LIN {X 0,Y 573.113,Z 1074.431,A -85,B 0,C 180,E1 -2244.193,E2 -2244.193} C_VEL
LIN {X 0,Y 573.004,Z 1079.986,A -85,B 0,C 180,E1 -2245.075,E2 -2245.075} C_VEL
LIN {X 0,Y 573.024,Z 1085.147,A -85,B 0,C 180,E1 -2246.132,E2 -2246.132} C_VEL
LIN {X 0,Y 572.99,Z 1087.788,A -85,B 0,C 180,E1 -2246.836,E2 -2246.836} C_VEL
LIN {X 0,Y 572.94,Z 1090.68,A -85,B 0,C 180,E1 -2247.891,E2 -2247.891} C_VEL
LIN {X 0,Y 572.944,Z 1091.936,A -85,B 0,C 180,E1 -2248.594,E2 -2248.594} C_VEL
LIN {X 0,Y 572.937,Z 1092.712,A -85,B 0,C 180,E1 -2249.297,E2 -2249.297} C_VEL
LIN {X 0,Y 572.935,Z 1093,A -85,B 0,C 180,E1 -2250,E2 -2250} C_VEL
LIN {X 0,Y 572.937,Z 1092.712,A -85,B 0,C 180,E1 -2250.703,E2 -2250.703} C_VEL
LIN {X 0,Y 572.944,Z 1091.936,A -85,B 0,C 180,E1 -2251.406,E2 -2251.406} C_VEL
LIN {X 0,Y 572.94,Z 1090.68,A -85,B 0,C 180,E1 -2252.109,E2 -2252.109} C_VEL
LIN {X 0,Y 572.99,Z 1087.788,A -85,B 0,C 180,E1 -2253.164,E2 -2253.164} C_VEL
LIN {X 0,Y 573.036,Z 1085.148,A -85,B 0,C 180,E1 -2253.868,E2 -2253.868} C_VEL
LIN {X 0,Y 573.004,Z 1079.986,A -85,B 0,C 180,E1 -2254.925,E2 -2254.925} C_VEL
LIN {X 0,Y 573.112,Z 1074.431,A -85,B 0,C 180,E1 -2255.806,E2 -2255.806} C_VEL
LIN {X 0,Y 573.155,Z 1067.55,A -85,B 0,C 180,E1 -2256.677,E2 -2256.677} C_VEL
LIN {X 0,Y 573.187,Z 1059.42,A -85,B 0,C 180,E1 -2257.485,E2 -2257.485} C_VEL
LIN {X 0,Y 573.256,Z 1051.769,A -85,B 0,C 180,E1 -2258.105,E2 -2258.105} C_VEL
LIN {X 0,Y 573.361,Z 1043.729,A -85,B 0,C 180,E1 -2258.636,E2 -2258.636} C_VEL
LIN {X 0,Y 573.393,Z 1035.4,A -85,B 0,C 180,E1 -2259.08,E2 -2259.08} C_VEL
LIN {X 0,Y 573.442,Z 1026.896,A -85,B 0,C 180,E1 -2259.434,E2 -2259.434} C_VEL
LIN {X 0,Y 573.468,Z 1016.757,A -85,B 0,C 180,E1 -2259.746,E2 -2259.746} C_VEL
LIN {X 0,Y 573.603,Z 1005.066,A -85,B 0,C 180,E1 -2259.966,E2 -2259.966} C_VEL
LIN {X 0,Y 573.476,Z 935.024,A -85,B 0,C 180,E1 -2260.842,E2 -2260.842} C_VEL
LIN {X 0,Y 573.182,Z 932.72,A -85,B 0,C 180,E1 -2260.883,E2 -2260.883} C_VEL
LIN {X 0,Y 573.294,Z 914.402,A -85,B 0,C 180,E1 -2263.83,E2 -2263.83} C_VEL
LIN {X 0,Y 573.477,Z 896.612,A -85,B 0,C 180,E1 -2266.725,E2 -2266.725} C_VEL
LIN {X 0,Y 573.619,Z 878.673,A -85,B 0,C 180,E1 -2269.69,E2 -2269.69} C_VEL
LIN {X 0,Y 573.625,Z 866.389,A -85,B 0,C 180,E1 -2271.754,E2 -2271.754} C_VEL
LIN {X 0,Y 573.2,Z 863.899,A -85,B 0,C 180,E1 -2272.197,E2 -2272.197} C_VEL
LIN {X 0,Y 573.186,Z 863.903,A -85,B 0,C 180,E1 -2274.861,E2 -2274.861} C_VEL
LIN {X 0,Y 573.182,Z 863.903,A -85,B 0,C 180,E1 -2276.979,E2 -2276.979} C_VEL
LIN {X 0,Y 573.193,Z 863.898,A -85,B 0,C 180,E1 -2279.479,E2 -2279.479} C_VEL
LIN {X 0,Y 573.218,Z 863.889,A -85,B 0,C 180,E1 -2282.223,E2 -2282.223} C_VEL
LIN {X 0,Y 573.212,Z 863.891,A -85,B 0,C 180,E1 -2284.768,E2 -2284.768} C_VEL
LIN {X 0,Y 573.184,Z 863.9,A -85,B 0,C 180,E1 -2287.812,E2 -2287.812} C_VEL
LIN {X 0,Y 573.197,Z 863.891,A -85,B 0,C 180,E1 -2290.529,E2 -2290.529} C_VEL
LIN {X 0,Y 573.183,Z 863.896,A -85,B 0,C 180,E1 -2293.364,E2 -2293.364} C_VEL
LIN {X 0,Y 573.191,Z 863.896,A -85,B 0,C 180,E1 -2296.337,E2 -2296.337} C_VEL
LIN {X 0,Y 573.183,Z 863.896,A -85,B 0,C 180,E1 -2298.539,E2 -2298.539} C_VEL
LIN {X 0,Y 573.174,Z 863.894,A -85,B 0,C 180,E1 -2301.293,E2 -2301.293} C_VEL
LIN {X 0,Y 573.178,Z 863.899,A -85,B 0,C 180,E1 -2304.023,E2 -2304.023} C_VEL
LIN {X 0,Y 573.22,Z 863.898,A -85,B 0,C 180,E1 -2306.515,E2 -2306.515} C_VEL
LIN {X 0,Y 573.198,Z 863.893,A -85,B 0,C 180,E1 -2309.123,E2 -2309.123} C_VEL
LIN {X 0,Y 573.19,Z 863.893,A -85,B 0,C 180,E1 -2311.983,E2 -2311.983} C_VEL
LIN {X 0,Y 573.194,Z 863.899,A -85,B 0,C 180,E1 -2314.587,E2 -2314.587} C_VEL
LIN {X 0,Y 573.191,Z 863.904,A -85,B 0,C 180,E1 -2316.899,E2 -2316.899} C_VEL
LIN {X 0,Y 573.223,Z 863.897,A -85,B 0,C 180,E1 -2319.173,E2 -2319.173} C_VEL
LIN {X 0,Y 573.189,Z 863.9,A -85,B 0,C 180,E1 -2321.41,E2 -2321.41} C_VEL
LIN {X 0,Y 573.247,Z 863.914,A -85,B 0,C 180,E1 -2322.52,E2 -2322.52} C_VEL
LIN {X 0,Y 573.186,Z 877.285,A -85,B 0,C 180,E1 -2325.444,E2 -2325.444} C_VEL
LIN {X 0,Y 573.114,Z 890.643,A -85,B 0,C 180,E1 -2328.327,E2 -2328.327} C_VEL
LIN {X 0,Y 573.113,Z 894.661,A -85,B 0,C 180,E1 -2329.188,E2 -2329.188} C_VEL
LIN {X 0,Y 573.677,Z 900.915,A -85,B 0,C 180,E1 -2329.281,E2 -2329.281} C_VEL
LIN {X 0,Y 573.529,Z 970.436,A -85,B 0,C 180,E1 -2330.167,E2 -2330.167} C_VEL
LIN {X 0,Y 573.478,Z 980.906,A -85,B 0,C 180,E1 -2330.411,E2 -2330.411} C_VEL
LIN {X 0,Y 573.381,Z 992.584,A -85,B 0,C 180,E1 -2330.832,E2 -2330.832} C_VEL
LIN {X 0,Y 573.369,Z 1003.02,A -85,B 0,C 180,E1 -2331.365,E2 -2331.365} C_VEL
LIN {X 0,Y 573.243,Z 1012.409,A -85,B 0,C 180,E1 -2331.984,E2 -2331.984} C_VEL
LIN {X 0,Y 573.188,Z 1021.892,A -85,B 0,C 180,E1 -2332.78,E2 -2332.78} C_VEL
LIN {X 0,Y 573.129,Z 1030.032,A -85,B 0,C 180,E1 -2333.664,E2 -2333.664} C_VEL
LIN {X 0,Y 573.051,Z 1036.508,A -85,B 0,C 180,E1 -2334.546,E2 -2334.546} C_VEL
LIN {X 0,Y 573.047,Z 1041.68,A -85,B 0,C 180,E1 -2335.428,E2 -2335.428} C_VEL
LIN {X 0,Y 573.025,Z 1046.439,A -85,B 0,C 180,E1 -2336.485,E2 -2336.485} C_VEL
LIN {X 0,Y 572.962,Z 1048.797,A -85,B 0,C 180,E1 -2337.188,E2 -2337.188} C_VEL
LIN {X 0,Y 572.94,Z 1050.597,A -85,B 0,C 180,E1 -2337.891,E2 -2337.891} C_VEL
LIN {X 0,Y 572.944,Z 1051.898,A -85,B 0,C 180,E1 -2338.595,E2 -2338.595} C_VEL
LIN {X 0,Y 572.936,Z 1052.709,A -85,B 0,C 180,E1 -2339.297,E2 -2339.297} C_VEL
LIN {X 0,Y 572.936,Z 1052.996,A -85,B 0,C 180,E1 -2340,E2 -2340} C_VEL
LIN {X 0,Y 572.937,Z 1052.75,A -85,B 0,C 180,E1 -2340.703,E2 -2340.703} C_VEL
LIN {X 0,Y 572.945,Z 1052.018,A -85,B 0,C 180,E1 -2341.406,E2 -2341.406} C_VEL
LIN {X 0,Y 572.941,Z 1050.801,A -85,B 0,C 180,E1 -2342.109,E2 -2342.109} C_VEL
LIN {X 0,Y 572.991,Z 1047.951,A -85,B 0,C 180,E1 -2343.164,E2 -2343.164} C_VEL
LIN {X 0,Y 573.033,Z 1043.853,A -85,B 0,C 180,E1 -2344.22,E2 -2344.22} C_VEL
LIN {X 0,Y 573.016,Z 1038.249,A -85,B 0,C 180,E1 -2345.278,E2 -2345.278} C_VEL
LIN {X 0,Y 573.145,Z 1032.173,A -85,B 0,C 180,E1 -2346.16,E2 -2346.16} C_VEL
LIN {X 0,Y 573.164,Z 1024.503,A -85,B 0,C 180,E1 -2347.044,E2 -2347.044} C_VEL
LIN {X 0,Y 573.237,Z 1015.883,A -85,B 0,C 180,E1 -2347.84,E2 -2347.84} C_VEL
LIN {X 0,Y 573.354,Z 1006.003,A -85,B 0,C 180,E1 -2348.548,E2 -2348.548} C_VEL
LIN {X 0,Y 573.379,Z 996.339,A -85,B 0,C 180,E1 -2349.08,E2 -2349.08} C_VEL
LIN {X 0,Y 573.411,Z 988.108,A -85,B 0,C 180,E1 -2349.435,E2 -2349.435} C_VEL
LIN {X 0,Y 573.475,Z 979.257,A -85,B 0,C 180,E1 -2349.724,E2 -2349.724} C_VEL
LIN {X 0,Y 573.546,Z 970.451,A -85,B 0,C 180,E1 -2349.923,E2 -2349.923} C_VEL
LIN {X 0,Y 573.521,Z 897.598,A -85,B 0,C 180,E1 -2350.854,E2 -2350.854} C_VEL
LIN {X 0,Y 573.113,Z 894.647,A -85,B 0,C 180,E1 -2350.905,E2 -2350.905} C_VEL
LIN {X 0,Y 573.165,Z 881.032,A -85,B 0,C 180,E1 -2353.834,E2 -2353.834} C_VEL
LIN {X 0,Y 573.155,Z 880.165,A -85,B 0,C 180,E1 -2354.022,E2 -2354.022} C_VEL
LIN {X 0,Y 572.495,Z 877.772,A -85,B 0,C 180,E1 -2354.558,E2 -2354.558} C_VEL
LIN {X 0,Y 566.909,Z 870.416,A -85,B 0,C 180,E1 -2356.327,E2 -2356.327} C_VEL
LIN {X 0,Y 566.259,Z 868.043,A -85,B 0,C 180,E1 -2356.873,E2 -2356.873} C_VEL
LIN {X 0,Y 566.195,Z 864.767,A -85,B 0,C 180,E1 -2357.612,E2 -2357.612} C_VEL
LIN {X 0,Y 566.151,Z 864.769,A -85,B 0,C 180,E1 -2360.34,E2 -2360.34} C_VEL
LIN {X 0,Y 566.132,Z 864.773,A -85,B 0,C 180,E1 -2362.634,E2 -2362.634} C_VEL
LIN {X 0,Y 566.164,Z 864.773,A -85,B 0,C 180,E1 -2365.018,E2 -2365.018} C_VEL
LIN {X 0,Y 566.161,Z 864.778,A -85,B 0,C 180,E1 -2367.342,E2 -2367.342} C_VEL
LIN {X 0,Y 566.147,Z 864.775,A -85,B 0,C 180,E1 -2369.772,E2 -2369.772} C_VEL
LIN {X 0,Y 566.176,Z 864.766,A -85,B 0,C 180,E1 -2372.425,E2 -2372.425} C_VEL
LIN {X 0,Y 566.162,Z 864.768,A -85,B 0,C 180,E1 -2374.987,E2 -2374.987} C_VEL
LIN {X 0,Y 566.181,Z 864.77,A -85,B 0,C 180,E1 -2377.463,E2 -2377.463} C_VEL
LIN {X 0,Y 566.159,Z 864.774,A -85,B 0,C 180,E1 -2380.204,E2 -2380.204} C_VEL
LIN {X 0,Y 566.144,Z 864.769,A -85,B 0,C 180,E1 -2383.06,E2 -2383.06} C_VEL
LIN {X 0,Y 566.146,Z 864.778,A -85,B 0,C 180,E1 -2386.055,E2 -2386.055} C_VEL
LIN {X 0,Y 566.135,Z 864.773,A -85,B 0,C 180,E1 -2388.857,E2 -2388.857} C_VEL
LIN {X 0,Y 566.158,Z 864.768,A -85,B 0,C 180,E1 -2391.449,E2 -2391.449} C_VEL
LIN {X 0,Y 566.159,Z 864.768,A -85,B 0,C 180,E1 -2393.793,E2 -2393.793} C_VEL
LIN {X 0,Y 566.198,Z 864.767,A -85,B 0,C 180,E1 -2396.269,E2 -2396.269} C_VEL
LIN {X 0,Y 566.172,Z 864.774,A -85,B 0,C 180,E1 -2398.928,E2 -2398.928} C_VEL
LIN {X 0,Y 566.143,Z 864.77,A -85,B 0,C 180,E1 -2401.854,E2 -2401.854} C_VEL
LIN {X 0,Y 566.171,Z 864.767,A -85,B 0,C 180,E1 -2404.249,E2 -2404.249} C_VEL
LIN {X 0,Y 566.149,Z 864.776,A -85,B 0,C 180,E1 -2407.367,E2 -2407.367} C_VEL
LIN {X 0,Y 566.159,Z 864.772,A -85,B 0,C 180,E1 -2409.661,E2 -2409.661} C_VEL
LIN {X 0,Y 566.164,Z 864.769,A -85,B 0,C 180,E1 -2411.921,E2 -2411.921} C_VEL
LIN {X 0,Y 566.182,Z 864.767,A -85,B 0,C 180,E1 -2414.89,E2 -2414.89} C_VEL
LIN {X 0,Y 566.159,Z 864.775,A -85,B 0,C 180,E1 -2417.817,E2 -2417.817} C_VEL
LIN {X 0,Y 566.132,Z 864.777,A -85,B 0,C 180,E1 -2419.991,E2 -2419.991} C_VEL
LIN {X 0,Y 566.183,Z 864.769,A -85,B 0,C 180,E1 -2422.152,E2 -2422.152} C_VEL
LIN {X 0,Y 566.247,Z 864.757,A -85,B 0,C 180,E1 -2425.016,E2 -2425.016} C_VEL
LIN {X 0,Y 566.279,Z 864.76,A -85,B 0,C 180,E1 -2427.866,E2 -2427.866} C_VEL
LIN {X 0,Y 566.288,Z 864.76,A -85,B 0,C 180,E1 -2430,E2 -2430} C_VEL
LIN {X 0,Y 566.239,Z 864.76,A -85,B 0,C 180,E1 -2432.846,E2 -2432.846} C_VEL
LIN {X 0,Y 566.222,Z 864.761,A -85,B 0,C 180,E1 -2435.699,E2 -2435.699} C_VEL
LIN {X 0,Y 566.187,Z 864.774,A -85,B 0,C 180,E1 -2438.567,E2 -2438.567} C_VEL
LIN {X 0,Y 566.194,Z 864.764,A -85,B 0,C 180,E1 -2441.455,E2 -2441.455} C_VEL
LIN {X 0,Y 566.18,Z 864.771,A -85,B 0,C 180,E1 -2444.482,E2 -2444.482} C_VEL
LIN {X 0,Y 566.174,Z 864.77,A -85,B 0,C 180,E1 -2447.333,E2 -2447.333} C_VEL
LIN {X 0,Y 566.175,Z 864.768,A -85,B 0,C 180,E1 -2449.582,E2 -2449.582} C_VEL
LIN {X 0,Y 566.143,Z 864.77,A -85,B 0,C 180,E1 -2451.865,E2 -2451.865} C_VEL
LIN {X 0,Y 566.149,Z 864.769,A -85,B 0,C 180,E1 -2454.183,E2 -2454.183} C_VEL
LIN {X 0,Y 566.17,Z 864.767,A -85,B 0,C 180,E1 -2456.65,E2 -2456.65} C_VEL
LIN {X 0,Y 566.149,Z 864.774,A -85,B 0,C 180,E1 -2459.772,E2 -2459.772} C_VEL
LIN {X 0,Y 566.141,Z 864.77,A -85,B 0,C 180,E1 -2462.419,E2 -2462.419} C_VEL
LIN {X 0,Y 566.163,Z 864.768,A -85,B 0,C 180,E1 -2464.986,E2 -2464.986} C_VEL
LIN {X 0,Y 566.158,Z 864.773,A -85,B 0,C 180,E1 -2467.464,E2 -2467.464} C_VEL
LIN {X 0,Y 566.161,Z 864.773,A -85,B 0,C 180,E1 -2470.203,E2 -2470.203} C_VEL
LIN {X 0,Y 566.143,Z 864.769,A -85,B 0,C 180,E1 -2473.06,E2 -2473.06} C_VEL
LIN {X 0,Y 566.146,Z 864.778,A -85,B 0,C 180,E1 -2476.055,E2 -2476.055} C_VEL
LIN {X 0,Y 566.136,Z 864.773,A -85,B 0,C 180,E1 -2478.856,E2 -2478.856} C_VEL
LIN {X 0,Y 566.158,Z 864.768,A -85,B 0,C 180,E1 -2481.449,E2 -2481.449} C_VEL
LIN {X 0,Y 566.138,Z 864.777,A -85,B 0,C 180,E1 -2484.306,E2 -2484.306} C_VEL
LIN {X 0,Y 566.165,Z 864.774,A -85,B 0,C 180,E1 -2486.894,E2 -2486.894} C_VEL
LIN {X 0,Y 566.151,Z 864.77,A -85,B 0,C 180,E1 -2489.405,E2 -2489.405} C_VEL
LIN {X 0,Y 566.143,Z 864.77,A -85,B 0,C 180,E1 -2491.853,E2 -2491.853} C_VEL
LIN {X 0,Y 566.171,Z 864.767,A -85,B 0,C 180,E1 -2494.248,E2 -2494.248} C_VEL
LIN {X 0,Y 566.148,Z 864.776,A -85,B 0,C 180,E1 -2497.367,E2 -2497.367} C_VEL
LIN {X 0,Y 566.157,Z 864.771,A -85,B 0,C 180,E1 -2499.66,E2 -2499.66} C_VEL
LIN {X 0,Y 566.163,Z 864.769,A -85,B 0,C 180,E1 -2501.92,E2 -2501.92} C_VEL
LIN {X 0,Y 566.174,Z 864.766,A -85,B 0,C 180,E1 -2504.151,E2 -2504.151} C_VEL
LIN {X 0,Y 566.157,Z 864.768,A -85,B 0,C 180,E1 -2506.357,E2 -2506.357} C_VEL
LIN {X 0,Y 566.199,Z 864.767,A -85,B 0,C 180,E1 -2509.269,E2 -2509.269} C_VEL
LIN {X 0,Y 566.181,Z 864.769,A -85,B 0,C 180,E1 -2512.152,E2 -2512.152} C_VEL
LIN {X 0,Y 566.246,Z 864.757,A -85,B 0,C 180,E1 -2515.015,E2 -2515.015} C_VEL
LIN {X 0,Y 566.278,Z 864.761,A -85,B 0,C 180,E1 -2517.866,E2 -2517.866} C_VEL
LIN {X 0,Y 566.286,Z 864.761,A -85,B 0,C 180,E1 -2520,E2 -2520} C_VEL
LIN {X 0,Y 566.237,Z 864.76,A -85,B 0,C 180,E1 -2522.845,E2 -2522.845} C_VEL
LIN {X 0,Y 566.22,Z 864.761,A -85,B 0,C 180,E1 -2525.698,E2 -2525.698} C_VEL
LIN {X 0,Y 566.184,Z 864.774,A -85,B 0,C 180,E1 -2528.566,E2 -2528.566} C_VEL
LIN {X 0,Y 566.191,Z 864.764,A -85,B 0,C 180,E1 -2531.455,E2 -2531.455} C_VEL
LIN {X 0,Y 566.205,Z 864.768,A -85,B 0,C 180,E1 -2534.493,E2 -2534.493} C_VEL
LIN {X 0,Y 566.171,Z 864.77,A -85,B 0,C 180,E1 -2537.332,E2 -2537.332} C_VEL
LIN {X 0,Y 566.171,Z 864.768,A -85,B 0,C 180,E1 -2539.582,E2 -2539.582} C_VEL
LIN {X 0,Y 566.14,Z 864.77,A -85,B 0,C 180,E1 -2541.864,E2 -2541.864} C_VEL
LIN {X 0,Y 566.146,Z 864.769,A -85,B 0,C 180,E1 -2544.183,E2 -2544.183} C_VEL
LIN {X 0,Y 566.166,Z 864.768,A -85,B 0,C 180,E1 -2546.65,E2 -2546.65} C_VEL
LIN {X 0,Y 566.145,Z 864.774,A -85,B 0,C 180,E1 -2549.772,E2 -2549.772} C_VEL
LIN {X 0,Y 566.137,Z 864.77,A -85,B 0,C 180,E1 -2552.419,E2 -2552.419} C_VEL
LIN {X 0,Y 566.16,Z 864.768,A -85,B 0,C 180,E1 -2554.986,E2 -2554.986} C_VEL
LIN {X 0,Y 566.156,Z 864.773,A -85,B 0,C 180,E1 -2557.464,E2 -2557.464} C_VEL
LIN {X 0,Y 566.157,Z 864.773,A -85,B 0,C 180,E1 -2560.203,E2 -2560.203} C_VEL
LIN {X 0,Y 566.141,Z 864.77,A -85,B 0,C 180,E1 -2563.06,E2 -2563.06} C_VEL
LIN {X 0,Y 566.143,Z 864.779,A -85,B 0,C 180,E1 -2566.054,E2 -2566.054} C_VEL
LIN {X 0,Y 566.132,Z 864.773,A -85,B 0,C 180,E1 -2568.856,E2 -2568.856} C_VEL
LIN {X 0,Y 566.155,Z 864.768,A -85,B 0,C 180,E1 -2571.449,E2 -2571.449} C_VEL
LIN {X 0,Y 566.135,Z 864.778,A -85,B 0,C 180,E1 -2574.306,E2 -2574.306} C_VEL
LIN {X 0,Y 566.16,Z 864.774,A -85,B 0,C 180,E1 -2576.894,E2 -2576.894} C_VEL
LIN {X 0,Y 566.147,Z 864.77,A -85,B 0,C 180,E1 -2579.405,E2 -2579.405} C_VEL
LIN {X 0,Y 566.138,Z 864.77,A -85,B 0,C 180,E1 -2581.853,E2 -2581.853} C_VEL
LIN {X 0,Y 566.167,Z 864.769,A -85,B 0,C 180,E1 -2584.248,E2 -2584.248} C_VEL
LIN {X 0,Y 566.155,Z 864.778,A -85,B 0,C 180,E1 -2587.367,E2 -2587.367} C_VEL
LIN {X 0,Y 566.203,Z 864.991,A -85,B 0,C 180,E1 -2587.706,E2 -2587.706} C_VEL
LIN {X 0,Y 566.808,Z 870.505,A -85,B 0,C 180,E1 -2588.675,E2 -2588.675} C_VEL
LIN {X 0,Y 566.569,Z 887.602,A -85,B 0,C 180,E1 -2591.56,E2 -2591.56} C_VEL
LIN {X 0,Y 566.37,Z 905.467,A -85,B 0,C 180,E1 -2594.526,E2 -2594.526} C_VEL
LIN {X 0,Y 566.196,Z 924.449,A -85,B 0,C 180,E1 -2597.636,E2 -2597.636} C_VEL
LIN {X 0,Y 566.143,Z 932.732,A -85,B 0,C 180,E1 -2598.982,E2 -2598.982} C_VEL
LIN {X 0,Y 566.664,Z 939.256,A -85,B 0,C 180,E1 -2599.08,E2 -2599.08} C_VEL
LIN {X 0,Y 566.574,Z 1009.129,A -85,B 0,C 180,E1 -2599.977,E2 -2599.977} C_VEL
LIN {X 0,Y 566.483,Z 1018.407,A -85,B 0,C 180,E1 -2600.178,E2 -2600.178} C_VEL
LIN {X 0,Y 566.455,Z 1026.888,A -85,B 0,C 180,E1 -2600.448,E2 -2600.448} C_VEL
LIN {X 0,Y 566.38,Z 1035.396,A -85,B 0,C 180,E1 -2600.807,E2 -2600.807} C_VEL
LIN {X 0,Y 566.346,Z 1043.727,A -85,B 0,C 180,E1 -2601.256,E2 -2601.256} C_VEL
LIN {X 0,Y 566.232,Z 1051.764,A -85,B 0,C 180,E1 -2601.794,E2 -2601.794} C_VEL
LIN {X 0,Y 566.146,Z 1059.414,A -85,B 0,C 180,E1 -2602.421,E2 -2602.421} C_VEL
LIN {X 0,Y 566.095,Z 1068.155,A -85,B 0,C 180,E1 -2603.309,E2 -2603.309} C_VEL
LIN {X 0,Y 566.057,Z 1074.432,A -85,B 0,C 180,E1 -2604.121,E2 -2604.121} C_VEL
LIN {X 0,Y 565.911,Z 1079.986,A -85,B 0,C 180,E1 -2605.013,E2 -2605.013} C_VEL
LIN {X 0,Y 565.934,Z 1085.147,A -85,B 0,C 180,E1 -2606.083,E2 -2606.083} C_VEL
LIN {X 0,Y 565.914,Z 1087.788,A -85,B 0,C 180,E1 -2606.796,E2 -2606.796} C_VEL
LIN {X 0,Y 565.841,Z 1090.68,A -85,B 0,C 180,E1 -2607.864,E2 -2607.864} C_VEL
LIN {X 0,Y 565.844,Z 1091.936,A -85,B 0,C 180,E1 -2608.576,E2 -2608.576} C_VEL
LIN {X 0,Y 565.837,Z 1092.711,A -85,B 0,C 180,E1 -2609.288,E2 -2609.288} C_VEL
LIN {X 0,Y 565.836,Z 1093,A -85,B 0,C 180,E1 -2610,E2 -2610} C_VEL
LIN {X 0,Y 565.837,Z 1092.711,A -85,B 0,C 180,E1 -2610.712,E2 -2610.712} C_VEL
LIN {X 0,Y 565.844,Z 1091.936,A -85,B 0,C 180,E1 -2611.423,E2 -2611.423} C_VEL
LIN {X 0,Y 565.84,Z 1090.681,A -85,B 0,C 180,E1 -2612.135,E2 -2612.135} C_VEL
LIN {X 0,Y 565.912,Z 1087.788,A -85,B 0,C 180,E1 -2613.204,E2 -2613.204} C_VEL
LIN {X 0,Y 565.944,Z 1085.148,A -85,B 0,C 180,E1 -2613.916,E2 -2613.916} C_VEL
LIN {X 0,Y 565.911,Z 1079.986,A -85,B 0,C 180,E1 -2614.987,E2 -2614.987} C_VEL
LIN {X 0,Y 566.082,Z 1073.188,A -85,B 0,C 180,E1 -2616.058,E2 -2616.058} C_VEL
LIN {X 0,Y 566.091,Z 1066.178,A -85,B 0,C 180,E1 -2616.907,E2 -2616.907} C_VEL
LIN {X 0,Y 566.145,Z 1058.407,A -85,B 0,C 180,E1 -2617.669,E2 -2617.669} C_VEL
LIN {X 0,Y 566.239,Z 1050.549,A -85,B 0,C 180,E1 -2618.296,E2 -2618.296} C_VEL
LIN {X 0,Y 566.354,Z 1040.735,A -85,B 0,C 180,E1 -2618.923,E2 -2618.923} C_VEL
LIN {X 0,Y 566.413,Z 1029.303,A -85,B 0,C 180,E1 -2619.463,E2 -2619.463} C_VEL
LIN {X 0,Y 566.505,Z 1019.249,A -85,B 0,C 180,E1 -2619.799,E2 -2619.799} C_VEL
LIN {X 0,Y 566.551,Z 1010.449,A -85,B 0,C 180,E1 -2620.001,E2 -2620.001} C_VEL
LIN {X 0,Y 566.645,Z 954.982,A -85,B 0,C 180,E1 -2620.722,E2 -2620.722} C_VEL
LIN {X 0,Y 566.639,Z 936.596,A -85,B 0,C 180,E1 -2620.954,E2 -2620.954} C_VEL
LIN {X 0,Y 566.146,Z 932.717,A -85,B 0,C 180,E1 -2621.02,E2 -2621.02} C_VEL
LIN {X 0,Y 566.268,Z 915.518,A -85,B 0,C 180,E1 -2623.822,E2 -2623.822} C_VEL
LIN {X 0,Y 566.439,Z 898.77,A -85,B 0,C 180,E1 -2626.581,E2 -2626.581} C_VEL
LIN {X 0,Y 566.664,Z 881.914,A -85,B 0,C 180,E1 -2629.394,E2 -2629.394} C_VEL
LIN {X 0,Y 566.77,Z 869.11,A -85,B 0,C 180,E1 -2631.564,E2 -2631.564} C_VEL
LIN {X 0,Y 566.178,Z 864.775,A -85,B 0,C 180,E1 -2632.343,E2 -2632.343} C_VEL
LIN {X 0,Y 566.139,Z 864.782,A -85,B 0,C 180,E1 -2635.013,E2 -2635.013} C_VEL
LIN {X 0,Y 566.155,Z 864.776,A -85,B 0,C 180,E1 -2637.342,E2 -2637.342} C_VEL
LIN {X 0,Y 566.142,Z 864.773,A -85,B 0,C 180,E1 -2639.772,E2 -2639.772} C_VEL
LIN {X 0,Y 566.169,Z 864.767,A -85,B 0,C 180,E1 -2642.424,E2 -2642.424} C_VEL
LIN {X 0,Y 566.158,Z 864.772,A -85,B 0,C 180,E1 -2644.986,E2 -2644.986} C_VEL
LIN {X 0,Y 566.152,Z 864.778,A -85,B 0,C 180,E1 -2647.464,E2 -2647.464} C_VEL
LIN {X 0,Y 566.154,Z 864.771,A -85,B 0,C 180,E1 -2650.204,E2 -2650.204} C_VEL
LIN {X 0,Y 566.135,Z 864.772,A -85,B 0,C 180,E1 -2653.06,E2 -2653.06} C_VEL
LIN {X 0,Y 566.142,Z 864.779,A -85,B 0,C 180,E1 -2656.055,E2 -2656.055} C_VEL
LIN {X 0,Y 566.131,Z 864.772,A -85,B 0,C 180,E1 -2658.857,E2 -2658.857} C_VEL
LIN {X 0,Y 566.158,Z 864.769,A -85,B 0,C 180,E1 -2661.449,E2 -2661.449} C_VEL
LIN {X 0,Y 566.133,Z 864.782,A -85,B 0,C 180,E1 -2664.306,E2 -2664.306} C_VEL
LIN {X 0,Y 566.159,Z 864.772,A -85,B 0,C 180,E1 -2666.894,E2 -2666.894} C_VEL
LIN {X 0,Y 566.145,Z 864.77,A -85,B 0,C 180,E1 -2669.405,E2 -2669.405} C_VEL
LIN {X 0,Y 566.137,Z 864.771,A -85,B 0,C 180,E1 -2671.854,E2 -2671.854} C_VEL
LIN {X 0,Y 566.166,Z 864.77,A -85,B 0,C 180,E1 -2674.249,E2 -2674.249} C_VEL
LIN {X 0,Y 566.144,Z 864.779,A -85,B 0,C 180,E1 -2676.725,E2 -2676.725} C_VEL
LIN {X 0,Y 566.187,Z 864.775,A -85,B 0,C 180,E1 -2678.902,E2 -2678.902} C_VEL
LIN {X 0,Y 566.165,Z 864.778,A -85,B 0,C 180,E1 -2681.171,E2 -2681.171} C_VEL
LIN {X 0,Y 566.232,Z 864.961,A -85,B 0,C 180,E1 -2682.53,E2 -2682.53} C_VEL
LIN {X 0,Y 566.156,Z 877.448,A -85,B 0,C 180,E1 -2685.294,E2 -2685.294} C_VEL
LIN {X 0,Y 566.053,Z 890.646,A -85,B 0,C 180,E1 -2688.179,E2 -2688.179} C_VEL
LIN {X 0,Y 566.052,Z 894.641,A -85,B 0,C 180,E1 -2689.047,E2 -2689.047} C_VEL
LIN {X 0,Y 566.699,Z 901.636,A -85,B 0,C 180,E1 -2689.156,E2 -2689.156} C_VEL
LIN {X 0,Y 566.557,Z 969.17,A -85,B 0,C 180,E1 -2690.022,E2 -2690.022} C_VEL
LIN {X 0,Y 566.515,Z 978.439,A -85,B 0,C 180,E1 -2690.224,E2 -2690.224} C_VEL
LIN {X 0,Y 566.408,Z 988.116,A -85,B 0,C 180,E1 -2690.538,E2 -2690.538} C_VEL
LIN {X 0,Y 566.411,Z 998.199,A -85,B 0,C 180,E1 -2690.988,E2 -2690.988} C_VEL
LIN {X 0,Y 566.282,Z 1008.722,A -85,B 0,C 180,E1 -2691.615,E2 -2691.615} C_VEL
LIN {X 0,Y 566.167,Z 1017.924,A -85,B 0,C 180,E1 -2692.332,E2 -2692.332} C_VEL
LIN {X 0,Y 566.101,Z 1025.875,A -85,B 0,C 180,E1 -2693.103,E2 -2693.103} C_VEL
LIN {X 0,Y 566.057,Z 1034.151,A -85,B 0,C 180,E1 -2694.121,E2 -2694.121} C_VEL
LIN {X 0,Y 565.912,Z 1039.765,A -85,B 0,C 180,E1 -2695.013,E2 -2695.013} C_VEL
LIN {X 0,Y 565.944,Z 1044.992,A -85,B 0,C 180,E1 -2696.084,E2 -2696.084} C_VEL
LIN {X 0,Y 565.881,Z 1048.799,A -85,B 0,C 180,E1 -2697.153,E2 -2697.153} C_VEL
LIN {X 0,Y 565.841,Z 1050.603,A -85,B 0,C 180,E1 -2697.865,E2 -2697.865} C_VEL
LIN {X 0,Y 565.843,Z 1051.904,A -85,B 0,C 180,E1 -2698.577,E2 -2698.577} C_VEL
LIN {X 0,Y 565.837,Z 1052.712,A -85,B 0,C 180,E1 -2699.289,E2 -2699.289} C_VEL
LIN {X 0,Y 565.837,Z 1052.996,A -85,B 0,C 180,E1 -2700,E2 -2700} C_VEL
LIN {X 0,Y 565.838,Z 1052.754,A -85,B 0,C 180,E1 -2700.712,E2 -2700.712} C_VEL
LIN {X 0,Y 565.845,Z 1052.022,A -85,B 0,C 180,E1 -2701.424,E2 -2701.424} C_VEL
LIN {X 0,Y 565.841,Z 1050.804,A -85,B 0,C 180,E1 -2702.136,E2 -2702.136} C_VEL
LIN {X 0,Y 565.913,Z 1047.953,A -85,B 0,C 180,E1 -2703.204,E2 -2703.204} C_VEL
LIN {X 0,Y 565.963,Z 1043.854,A -85,B 0,C 180,E1 -2704.273,E2 -2704.273} C_VEL
LIN {X 0,Y 565.946,Z 1038.246,A -85,B 0,C 180,E1 -2705.344,E2 -2705.344} C_VEL
LIN {X 0,Y 566.084,Z 1032.171,A -85,B 0,C 180,E1 -2706.237,E2 -2706.237} C_VEL
LIN {X 0,Y 566.116,Z 1024.503,A -85,B 0,C 180,E1 -2707.132,E2 -2707.132} C_VEL
LIN {X 0,Y 566.175,Z 1015.878,A -85,B 0,C 180,E1 -2707.938,E2 -2707.938} C_VEL
LIN {X 0,Y 566.328,Z 1006.002,A -85,B 0,C 180,E1 -2708.654,E2 -2708.654} C_VEL
LIN {X 0,Y 566.365,Z 996.332,A -85,B 0,C 180,E1 -2709.194,E2 -2709.194} C_VEL
LIN {X 0,Y 566.447,Z 986.892,A -85,B 0,C 180,E1 -2709.598,E2 -2709.598} C_VEL
LIN {X 0,Y 566.506,Z 976.737,A -85,B 0,C 180,E1 -2709.912,E2 -2709.912} C_VEL
LIN {X 0,Y 566.596,Z 965.018,A -85,B 0,C 180,E1 -2710.136,E2 -2710.136} C_VEL
LIN {X 0,Y 566.639,Z 898.908,A -85,B 0,C 180,E1 -2710.97,E2 -2710.97} C_VEL
LIN {X 0,Y 566.045,Z 894.625,A -85,B 0,C 180,E1 -2711.047,E2 -2711.047} C_VEL
LIN {X 0,Y 566.118,Z 880.858,A -85,B 0,C 180,E1 -2714.047,E2 -2714.047} C_VEL
LIN {X 0,Y 566.259,Z 868.043,A -85,B 0,C 180,E1 -2716.873,E2 -2716.873} C_VEL
LIN {X 0,Y 565.931,Z 866.698,A -85,B 0,C 180,E1 -2717.242,E2 -2717.242} C_VEL
LIN {X 0,Y 564.573,Z 865.564,A -85,B 0,C 180,E1 -2717.812,E2 -2717.812} C_VEL
LIN {X 0,Y 562.707,Z 865.21,A -85,B 0,C 180,E1 -2718.385,E2 -2718.385} C_VEL
LIN {X 0,Y 560.273,Z 865.509,A -85,B 0,C 180,E1 -2719.175,E2 -2719.175} C_VEL
LIN {X 0,Y 559.217,Z 865.638,A -85,B 0,C 180,E1 -2719.783,E2 -2719.783} C_VEL
LIN {X 0,Y 559.123,Z 865.644,A -85,B 0,C 180,E1 -2719.989,E2 -2719.989} C_VEL
LIN {X 0,Y 559.098,Z 865.647,A -85,B 0,C 180,E1 -2722.155,E2 -2722.155} C_VEL
LIN {X 0,Y 559.131,Z 865.652,A -85,B 0,C 180,E1 -2725.176,E2 -2725.176} C_VEL
LIN {X 0,Y 559.101,Z 865.652,A -85,B 0,C 180,E1 -2727.717,E2 -2727.717} C_VEL
LIN {X 0,Y 559.093,Z 865.649,A -85,B 0,C 180,E1 -2730.187,E2 -2730.187} C_VEL
LIN {X 0,Y 559.135,Z 865.643,A -85,B 0,C 180,E1 -2732.717,E2 -2732.717} C_VEL
LIN {X 0,Y 559.115,Z 865.649,A -85,B 0,C 180,E1 -2735.326,E2 -2735.326} C_VEL
LIN {X 0,Y 559.115,Z 865.653,A -85,B 0,C 180,E1 -2738.02,E2 -2738.02} C_VEL
LIN {X 0,Y 559.093,Z 865.648,A -85,B 0,C 180,E1 -2740.819,E2 -2740.819} C_VEL
LIN {X 0,Y 559.1,Z 865.652,A -85,B 0,C 180,E1 -2743.739,E2 -2743.739} C_VEL
LIN {X 0,Y 559.093,Z 865.658,A -85,B 0,C 180,E1 -2746.261,E2 -2746.261} C_VEL
LIN {X 0,Y 559.092,Z 865.648,A -85,B 0,C 180,E1 -2749.182,E2 -2749.182} C_VEL
LIN {X 0,Y 559.099,Z 865.65,A -85,B 0,C 180,E1 -2751.98,E2 -2751.98} C_VEL
LIN {X 0,Y 559.121,Z 865.652,A -85,B 0,C 180,E1 -2754.79,E2 -2754.79} C_VEL
LIN {X 0,Y 559.138,Z 865.643,A -85,B 0,C 180,E1 -2757.368,E2 -2757.368} C_VEL
LIN {X 0,Y 559.098,Z 865.648,A -85,B 0,C 180,E1 -2760.153,E2 -2760.153} C_VEL
LIN {X 0,Y 559.114,Z 865.652,A -85,B 0,C 180,E1 -2763.185,E2 -2763.185} C_VEL
LIN {X 0,Y 559.089,Z 865.652,A -85,B 0,C 180,E1 -2765.492,E2 -2765.492} C_VEL
LIN {X 0,Y 559.14,Z 865.643,A -85,B 0,C 180,E1 -2768.456,E2 -2768.456} C_VEL
LIN {X 0,Y 559.138,Z 865.647,A -85,B 0,C 180,E1 -2770.925,E2 -2770.925} C_VEL
LIN {X 0,Y 559.136,Z 865.645,A -85,B 0,C 180,E1 -2773.947,E2 -2773.947} C_VEL
LIN {X 0,Y 559.145,Z 865.643,A -85,B 0,C 180,E1 -2776.184,E2 -2776.184} C_VEL
LIN {X 0,Y 559.158,Z 865.642,A -85,B 0,C 180,E1 -2779.133,E2 -2779.133} C_VEL
LIN {X 0,Y 559.138,Z 865.649,A -85,B 0,C 180,E1 -2782.053,E2 -2782.053} C_VEL
LIN {X 0,Y 559.224,Z 865.632,A -85,B 0,C 180,E1 -2784.953,E2 -2784.953} C_VEL
LIN {X 0,Y 559.249,Z 865.635,A -85,B 0,C 180,E1 -2787.84,E2 -2787.84} C_VEL
LIN {X 0,Y 559.256,Z 865.636,A -85,B 0,C 180,E1 -2790,E2 -2790} C_VEL
LIN {X 0,Y 559.206,Z 865.635,A -85,B 0,C 180,E1 -2792.882,E2 -2792.882} C_VEL
LIN {X 0,Y 559.193,Z 865.637,A -85,B 0,C 180,E1 -2795.771,E2 -2795.771} C_VEL
LIN {X 0,Y 559.152,Z 865.649,A -85,B 0,C 180,E1 -2798.675,E2 -2798.675} C_VEL
LIN {X 0,Y 559.134,Z 865.643,A -85,B 0,C 180,E1 -2801.602,E2 -2801.602} C_VEL
LIN {X 0,Y 559.138,Z 865.649,A -85,B 0,C 180,E1 -2804.568,E2 -2804.568} C_VEL
LIN {X 0,Y 559.123,Z 865.646,A -85,B 0,C 180,E1 -2807.558,E2 -2807.558} C_VEL
LIN {X 0,Y 559.138,Z 865.643,A -85,B 0,C 180,E1 -2809.839,E2 -2809.839} C_VEL
LIN {X 0,Y 559.1,Z 865.647,A -85,B 0,C 180,E1 -2812.155,E2 -2812.155} C_VEL
LIN {X 0,Y 559.122,Z 865.654,A -85,B 0,C 180,E1 -2815.173,E2 -2815.173} C_VEL
LIN {X 0,Y 559.103,Z 865.652,A -85,B 0,C 180,E1 -2817.717,E2 -2817.717} C_VEL
LIN {X 0,Y 559.095,Z 865.648,A -85,B 0,C 180,E1 -2820.187,E2 -2820.187} C_VEL
LIN {X 0,Y 559.1,Z 865.647,A -85,B 0,C 180,E1 -2822.719,E2 -2822.719} C_VEL
LIN {X 0,Y 559.117,Z 865.649,A -85,B 0,C 180,E1 -2825.325,E2 -2825.325} C_VEL
LIN {X 0,Y 559.094,Z 865.655,A -85,B 0,C 180,E1 -2828.021,E2 -2828.021} C_VEL
LIN {X 0,Y 559.094,Z 865.648,A -85,B 0,C 180,E1 -2830.818,E2 -2830.818} C_VEL
LIN {X 0,Y 559.095,Z 865.653,A -85,B 0,C 180,E1 -2833.739,E2 -2833.739} C_VEL
LIN {X 0,Y 559.093,Z 865.657,A -85,B 0,C 180,E1 -2836.261,E2 -2836.261} C_VEL
LIN {X 0,Y 559.093,Z 865.648,A -85,B 0,C 180,E1 -2839.181,E2 -2839.181} C_VEL
LIN {X 0,Y 559.093,Z 865.651,A -85,B 0,C 180,E1 -2841.979,E2 -2841.979} C_VEL
LIN {X 0,Y 559.121,Z 865.651,A -85,B 0,C 180,E1 -2844.789,E2 -2844.789} C_VEL
LIN {X 0,Y 559.139,Z 865.643,A -85,B 0,C 180,E1 -2847.368,E2 -2847.368} C_VEL
LIN {X 0,Y 559.098,Z 865.649,A -85,B 0,C 180,E1 -2850.152,E2 -2850.152} C_VEL
LIN {X 0,Y 559.114,Z 865.652,A -85,B 0,C 180,E1 -2853.185,E2 -2853.185} C_VEL
LIN {X 0,Y 559.089,Z 865.652,A -85,B 0,C 180,E1 -2855.491,E2 -2855.491} C_VEL
LIN {X 0,Y 559.14,Z 865.643,A -85,B 0,C 180,E1 -2858.456,E2 -2858.456} C_VEL
LIN {X 0,Y 559.137,Z 865.647,A -85,B 0,C 180,E1 -2860.925,E2 -2860.925} C_VEL
LIN {X 0,Y 559.144,Z 865.649,A -85,B 0,C 180,E1 -2863.196,E2 -2863.196} C_VEL
LIN {X 0,Y 559.14,Z 865.643,A -85,B 0,C 180,E1 -2866.183,E2 -2866.183} C_VEL
LIN {X 0,Y 559.157,Z 865.643,A -85,B 0,C 180,E1 -2869.132,E2 -2869.132} C_VEL
LIN {X 0,Y 559.136,Z 865.648,A -85,B 0,C 180,E1 -2872.052,E2 -2872.052} C_VEL
LIN {X 0,Y 559.222,Z 865.632,A -85,B 0,C 180,E1 -2874.953,E2 -2874.953} C_VEL
LIN {X 0,Y 559.248,Z 865.636,A -85,B 0,C 180,E1 -2877.839,E2 -2877.839} C_VEL
LIN {X 0,Y 559.254,Z 865.636,A -85,B 0,C 180,E1 -2880,E2 -2880} C_VEL
LIN {X 0,Y 559.204,Z 865.636,A -85,B 0,C 180,E1 -2882.881,E2 -2882.881} C_VEL
LIN {X 0,Y 559.191,Z 865.637,A -85,B 0,C 180,E1 -2885.77,E2 -2885.77} C_VEL
LIN {X 0,Y 559.15,Z 865.649,A -85,B 0,C 180,E1 -2888.675,E2 -2888.675} C_VEL
LIN {X 0,Y 559.131,Z 865.643,A -85,B 0,C 180,E1 -2891.602,E2 -2891.602} C_VEL
LIN {X 0,Y 559.155,Z 865.647,A -85,B 0,C 180,E1 -2894.576,E2 -2894.576} C_VEL
LIN {X 0,Y 559.12,Z 865.646,A -85,B 0,C 180,E1 -2897.558,E2 -2897.558} C_VEL
LIN {X 0,Y 559.135,Z 865.643,A -85,B 0,C 180,E1 -2899.838,E2 -2899.838} C_VEL
LIN {X 0,Y 559.097,Z 865.647,A -85,B 0,C 180,E1 -2902.154,E2 -2902.154} C_VEL
LIN {X 0,Y 559.118,Z 865.655,A -85,B 0,C 180,E1 -2905.173,E2 -2905.173} C_VEL
LIN {X 0,Y 559.099,Z 865.652,A -85,B 0,C 180,E1 -2907.716,E2 -2907.716} C_VEL
LIN {X 0,Y 559.091,Z 865.649,A -85,B 0,C 180,E1 -2910.186,E2 -2910.186} C_VEL
LIN {X 0,Y 559.096,Z 865.648,A -85,B 0,C 180,E1 -2912.719,E2 -2912.719} C_VEL
LIN {X 0,Y 559.113,Z 865.65,A -85,B 0,C 180,E1 -2915.325,E2 -2915.325} C_VEL
LIN {X 0,Y 559.094,Z 865.655,A -85,B 0,C 180,E1 -2918.02,E2 -2918.02} C_VEL
LIN {X 0,Y 559.09,Z 865.648,A -85,B 0,C 180,E1 -2920.818,E2 -2920.818} C_VEL
LIN {X 0,Y 559.097,Z 865.653,A -85,B 0,C 180,E1 -2923.738,E2 -2923.738} C_VEL
LIN {X 0,Y 559.09,Z 865.657,A -85,B 0,C 180,E1 -2926.261,E2 -2926.261} C_VEL
LIN {X 0,Y 559.089,Z 865.648,A -85,B 0,C 180,E1 -2929.181,E2 -2929.181} C_VEL
LIN {X 0,Y 559.089,Z 865.652,A -85,B 0,C 180,E1 -2931.979,E2 -2931.979} C_VEL
LIN {X 0,Y 559.117,Z 865.651,A -85,B 0,C 180,E1 -2934.789,E2 -2934.789} C_VEL
LIN {X 0,Y 559.134,Z 865.644,A -85,B 0,C 180,E1 -2937.368,E2 -2937.368} C_VEL
LIN {X 0,Y 559.094,Z 865.649,A -85,B 0,C 180,E1 -2940.152,E2 -2940.152} C_VEL
LIN {X 0,Y 559.11,Z 865.654,A -85,B 0,C 180,E1 -2943.185,E2 -2943.185} C_VEL
LIN {X 0,Y 559.086,Z 865.655,A -85,B 0,C 180,E1 -2945.491,E2 -2945.491} C_VEL
LIN {X 0,Y 559.153,Z 865.829,A -85,B 0,C 180,E1 -2947.556,E2 -2947.556} C_VEL
LIN {X 0,Y 559.866,Z 870.486,A -85,B 0,C 180,E1 -2948.395,E2 -2948.395} C_VEL
LIN {X 0,Y 559.597,Z 887.602,A -85,B 0,C 180,E1 -2951.321,E2 -2951.321} C_VEL
LIN {X 0,Y 559.365,Z 904.351,A -85,B 0,C 180,E1 -2954.141,E2 -2954.141} C_VEL
LIN {X 0,Y 559.163,Z 922.216,A -85,B 0,C 180,E1 -2957.109,E2 -2957.109} C_VEL
LIN {X 0,Y 559.115,Z 932.672,A -85,B 0,C 180,E1 -2958.832,E2 -2958.832} C_VEL
LIN {X 0,Y 559.707,Z 939.696,A -85,B 0,C 180,E1 -2958.948,E2 -2958.948} C_VEL
LIN {X 0,Y 559.598,Z 1009.129,A -85,B 0,C 180,E1 -2959.85,E2 -2959.85} C_VEL
LIN {X 0,Y 559.497,Z 1018.407,A -85,B 0,C 180,E1 -2960.054,E2 -2960.054} C_VEL
LIN {X 0,Y 559.472,Z 1026.887,A -85,B 0,C 180,E1 -2960.327,E2 -2960.327} C_VEL
LIN {X 0,Y 559.379,Z 1035.397,A -85,B 0,C 180,E1 -2960.691,E2 -2960.691} C_VEL
LIN {X 0,Y 559.328,Z 1043.728,A -85,B 0,C 180,E1 -2961.146,E2 -2961.146} C_VEL
LIN {X 0,Y 559.184,Z 1051.766,A -85,B 0,C 180,E1 -2961.689,E2 -2961.689} C_VEL
LIN {X 0,Y 559.094,Z 1060.428,A -85,B 0,C 180,E1 -2962.415,E2 -2962.415} C_VEL
LIN {X 0,Y 559.031,Z 1068.753,A -85,B 0,C 180,E1 -2963.299,E2 -2963.299} C_VEL
LIN {X 0,Y 559.004,Z 1074.432,A -85,B 0,C 180,E1 -2964.046,E2 -2964.046} C_VEL
LIN {X 0,Y 558.825,Z 1079.987,A -85,B 0,C 180,E1 -2964.949,E2 -2964.949} C_VEL
LIN {X 0,Y 558.851,Z 1085.147,A -85,B 0,C 180,E1 -2966.034,E2 -2966.034} C_VEL
LIN {X 0,Y 558.84,Z 1087.788,A -85,B 0,C 180,E1 -2966.756,E2 -2966.756} C_VEL
LIN {X 0,Y 558.746,Z 1090.681,A -85,B 0,C 180,E1 -2967.837,E2 -2967.837} C_VEL
LIN {X 0,Y 558.744,Z 1091.935,A -85,B 0,C 180,E1 -2968.558,E2 -2968.558} C_VEL
LIN {X 0,Y 558.737,Z 1092.71,A -85,B 0,C 180,E1 -2969.279,E2 -2969.279} C_VEL
LIN {X 0,Y 558.737,Z 1093,A -85,B 0,C 180,E1 -2970,E2 -2970} C_VEL
LIN {X 0,Y 558.737,Z 1092.71,A -85,B 0,C 180,E1 -2970.721,E2 -2970.721} C_VEL
LIN {X 0,Y 558.744,Z 1091.935,A -85,B 0,C 180,E1 -2971.441,E2 -2971.441} C_VEL
LIN {X 0,Y 558.746,Z 1090.681,A -85,B 0,C 180,E1 -2972.162,E2 -2972.162} C_VEL
LIN {X 0,Y 558.835,Z 1087.788,A -85,B 0,C 180,E1 -2973.244,E2 -2973.244} C_VEL
LIN {X 0,Y 558.859,Z 1085.148,A -85,B 0,C 180,E1 -2973.966,E2 -2973.966} C_VEL
LIN {X 0,Y 558.825,Z 1079.986,A -85,B 0,C 180,E1 -2975.05,E2 -2975.05} C_VEL
LIN {X 0,Y 559.018,Z 1073.188,A -85,B 0,C 180,E1 -2976.134,E2 -2976.134} C_VEL
LIN {X 0,Y 559.035,Z 1065.746,A -85,B 0,C 180,E1 -2977.04,E2 -2977.04} C_VEL
LIN {X 0,Y 559.118,Z 1058.408,A -85,B 0,C 180,E1 -2977.766,E2 -2977.766} C_VEL
LIN {X 0,Y 559.223,Z 1050.548,A -85,B 0,C 180,E1 -2978.401,E2 -2978.401} C_VEL
LIN {X 0,Y 559.318,Z 1040.733,A -85,B 0,C 180,E1 -2979.037,E2 -2979.037} C_VEL
LIN {X 0,Y 559.43,Z 1029.304,A -85,B 0,C 180,E1 -2979.582,E2 -2979.582} C_VEL
LIN {X 0,Y 559.52,Z 1019.249,A -85,B 0,C 180,E1 -2979.923,E2 -2979.923} C_VEL
LIN {X 0,Y 559.561,Z 1010.448,A -85,B 0,C 180,E1 -2980.127,E2 -2980.127} C_VEL
LIN {X 0,Y 559.707,Z 963.925,A -85,B 0,C 180,E1 -2980.742,E2 -2980.742} C_VEL
LIN {X 0,Y 559.613,Z 936.673,A -85,B 0,C 180,E1 -2981.093,E2 -2981.093} C_VEL
LIN {X 0,Y 559.107,Z 932.701,A -85,B 0,C 180,E1 -2981.164,E2 -2981.164} C_VEL
LIN {X 0,Y 559.244,Z 915.518,A -85,B 0,C 180,E1 -2983.999,E2 -2983.999} C_VEL
LIN {X 0,Y 559.474,Z 897.223,A -85,B 0,C 180,E1 -2987.054,E2 -2987.054} C_VEL
LIN {X 0,Y 559.73,Z 879.788,A -85,B 0,C 180,E1 -2990.008,E2 -2990.008} C_VEL
LIN {X 0,Y 559.701,Z 869.021,A -85,B 0,C 180,E1 -2991.866,E2 -2991.866} C_VEL
LIN {X 0,Y 559.131,Z 865.653,A -85,B 0,C 180,E1 -2992.494,E2 -2992.494} C_VEL
LIN {X 0,Y 559.097,Z 865.656,A -85,B 0,C 180,E1 -2995.302,E2 -2995.302} C_VEL
LIN {X 0,Y 559.097,Z 865.651,A -85,B 0,C 180,E1 -2997.717,E2 -2997.717} C_VEL
LIN {X 0,Y 559.089,Z 865.649,A -85,B 0,C 180,E1 -3000.187,E2 -3000.187} C_VEL
LIN {X 0,Y 559.13,Z 865.646,A -85,B 0,C 180,E1 -3002.717,E2 -3002.717} C_VEL
LIN {X 0,Y 559.111,Z 865.655,A -85,B 0,C 180,E1 -3005.325,E2 -3005.325} C_VEL
LIN {X 0,Y 559.088,Z 865.653,A -85,B 0,C 180,E1 -3008.021,E2 -3008.021} C_VEL
LIN {X 0,Y 559.087,Z 865.649,A -85,B 0,C 180,E1 -3010.819,E2 -3010.819} C_VEL
LIN {X 0,Y 559.087,Z 865.658,A -85,B 0,C 180,E1 -3013.739,E2 -3013.739} C_VEL
LIN {X 0,Y 559.089,Z 865.654,A -85,B 0,C 180,E1 -3016.261,E2 -3016.261} C_VEL
LIN {X 0,Y 559.088,Z 865.649,A -85,B 0,C 180,E1 -3019.182,E2 -3019.182} C_VEL
LIN {X 0,Y 559.092,Z 865.655,A -85,B 0,C 180,E1 -3021.979,E2 -3021.979} C_VEL
LIN {X 0,Y 559.116,Z 865.649,A -85,B 0,C 180,E1 -3024.79,E2 -3024.79} C_VEL
LIN {X 0,Y 559.133,Z 865.644,A -85,B 0,C 180,E1 -3027.368,E2 -3027.368} C_VEL
LIN {X 0,Y 559.093,Z 865.652,A -85,B 0,C 180,E1 -3030.153,E2 -3030.153} C_VEL
LIN {X 0,Y 559.107,Z 865.65,A -85,B 0,C 180,E1 -3033.186,E2 -3033.186} C_VEL
LIN {X 0,Y 559.084,Z 865.652,A -85,B 0,C 180,E1 -3035.492,E2 -3035.492} C_VEL
LIN {X 0,Y 559.154,Z 865.647,A -85,B 0,C 180,E1 -3038.623,E2 -3038.623} C_VEL
LIN {X 0,Y 559.133,Z 865.653,A -85,B 0,C 180,E1 -3040.925,E2 -3040.925} C_VEL
LIN {X 0,Y 559.168,Z 865.833,A -85,B 0,C 180,E1 -3042.499,E2 -3042.499} C_VEL
LIN {X 0,Y 559.125,Z 877.284,A -85,B 0,C 180,E1 -3045.068,E2 -3045.068} C_VEL
LIN {X 0,Y 558.994,Z 888.978,A -85,B 0,C 180,E1 -3047.659,E2 -3047.659} C_VEL
LIN {X 0,Y 558.996,Z 894.846,A -85,B 0,C 180,E1 -3048.917,E2 -3048.917} C_VEL
LIN {X 0,Y 559.741,Z 901.021,A -85,B 0,C 180,E1 -3049.011,E2 -3049.011} C_VEL
LIN {X 0,Y 559.583,Z 969.203,A -85,B 0,C 180,E1 -3049.896,E2 -3049.896} C_VEL
LIN {X 0,Y 559.53,Z 978.461,A -85,B 0,C 180,E1 -3050.101,E2 -3050.101} C_VEL
LIN {X 0,Y 559.414,Z 988.134,A -85,B 0,C 180,E1 -3050.418,E2 -3050.418} C_VEL
LIN {X 0,Y 559.383,Z 998.214,A -85,B 0,C 180,E1 -3050.874,E2 -3050.874} C_VEL
LIN {X 0,Y 559.266,Z 1008.726,A -85,B 0,C 180,E1 -3051.509,E2 -3051.509} C_VEL
LIN {X 0,Y 559.121,Z 1017.934,A -85,B 0,C 180,E1 -3052.234,E2 -3052.234} C_VEL
LIN {X 0,Y 559.068,Z 1025.368,A -85,B 0,C 180,E1 -3052.96,E2 -3052.96} C_VEL
LIN {X 0,Y 559.007,Z 1032.839,A -85,B 0,C 180,E1 -3053.866,E2 -3053.866} C_VEL
LIN {X 0,Y 558.826,Z 1039.767,A -85,B 0,C 180,E1 -3054.95,E2 -3054.95} C_VEL
LIN {X 0,Y 558.859,Z 1045,A -85,B 0,C 180,E1 -3056.034,E2 -3056.034} C_VEL
LIN {X 0,Y 558.804,Z 1048.802,A -85,B 0,C 180,E1 -3057.117,E2 -3057.117} C_VEL
LIN {X 0,Y 558.747,Z 1050.608,A -85,B 0,C 180,E1 -3057.838,E2 -3057.838} C_VEL
LIN {X 0,Y 558.743,Z 1051.909,A -85,B 0,C 180,E1 -3058.559,E2 -3058.559} C_VEL
LIN {X 0,Y 558.737,Z 1052.714,A -85,B 0,C 180,E1 -3059.28,E2 -3059.28} C_VEL
LIN {X 0,Y 558.738,Z 1052.996,A -85,B 0,C 180,E1 -3060,E2 -3060} C_VEL
LIN {X 0,Y 558.738,Z 1052.757,A -85,B 0,C 180,E1 -3060.721,E2 -3060.721} C_VEL
LIN {X 0,Y 558.745,Z 1052.026,A -85,B 0,C 180,E1 -3061.442,E2 -3061.442} C_VEL
LIN {X 0,Y 558.747,Z 1050.807,A -85,B 0,C 180,E1 -3062.163,E2 -3062.163} C_VEL
LIN {X 0,Y 558.836,Z 1047.955,A -85,B 0,C 180,E1 -3063.245,E2 -3063.245} C_VEL
LIN {X 0,Y 558.894,Z 1043.854,A -85,B 0,C 180,E1 -3064.327,E2 -3064.327} C_VEL
LIN {X 0,Y 558.881,Z 1038.242,A -85,B 0,C 180,E1 -3065.412,E2 -3065.412} C_VEL
LIN {X 0,Y 559.006,Z 1032.167,A -85,B 0,C 180,E1 -3066.316,E2 -3066.316} C_VEL
LIN {X 0,Y 559.056,Z 1024.502,A -85,B 0,C 180,E1 -3067.222,E2 -3067.222} C_VEL
LIN {X 0,Y 559.142,Z 1015.872,A -85,B 0,C 180,E1 -3068.039,E2 -3068.039} C_VEL
LIN {X 0,Y 559.32,Z 1006,A -85,B 0,C 180,E1 -3068.764,E2 -3068.764} C_VEL
LIN {X 0,Y 559.37,Z 996.324,A -85,B 0,C 180,E1 -3069.31,E2 -3069.31} C_VEL
LIN {X 0,Y 559.455,Z 986.876,A -85,B 0,C 180,E1 -3069.719,E2 -3069.719} C_VEL
LIN {X 0,Y 559.518,Z 976.714,A -85,B 0,C 180,E1 -3070.037,E2 -3070.037} C_VEL
LIN {X 0,Y 559.626,Z 964.973,A -85,B 0,C 180,E1 -3070.264,E2 -3070.264} C_VEL
LIN {X 0,Y 559.552,Z 898.727,A -85,B 0,C 180,E1 -3071.113,E2 -3071.113} C_VEL
LIN {X 0,Y 558.976,Z 894.639,A -85,B 0,C 180,E1 -3071.185,E2 -3071.185} C_VEL
LIN {X 0,Y 559.06,Z 882.698,A -85,B 0,C 180,E1 -3073.819,E2 -3073.819} C_VEL
LIN {X 0,Y 559.216,Z 868.846,A -85,B 0,C 180,E1 -3076.91,E2 -3076.91} C_VEL
LIN {X 0,Y 559.16,Z 865.643,A -85,B 0,C 180,E1 -3077.652,E2 -3077.652} C_VEL
LIN {X 0,Y 559.123,Z 865.644,A -85,B 0,C 180,E1 -3079.989,E2 -3079.989} C_VEL
LIN {X 0,Y 558.426,Z 865.735,A -85,B 0,C 180,E1 -3080.59,E2 -3080.59} C_VEL
LIN {X 0,Y 555.535,Z 866.095,A -85,B 0,C 180,E1 -3081.565,E2 -3081.565} C_VEL
LIN {X 0,Y 553.121,Z 866.394,A -85,B 0,C 180,E1 -3082.35,E2 -3082.35} C_VEL
LIN {X 0,Y 552.109,Z 866.525,A -85,B 0,C 180,E1 -3082.956,E2 -3082.956} C_VEL
LIN {X 0,Y 552.039,Z 866.535,A -85,B 0,C 180,E1 -3083.161,E2 -3083.161} C_VEL
LIN {X 0,Y 552.069,Z 866.528,A -85,B 0,C 180,E1 -3085.648,E2 -3085.648} C_VEL
LIN {X 0,Y 552.072,Z 866.523,A -85,B 0,C 180,E1 -3088.552,E2 -3088.552} C_VEL
LIN {X 0,Y 552.094,Z 866.529,A -85,B 0,C 180,E1 -3091.472,E2 -3091.472} C_VEL
LIN {X 0,Y 552.095,Z 866.523,A -85,B 0,C 180,E1 -3094.164,E2 -3094.164} C_VEL
LIN {X 0,Y 552.049,Z 866.525,A -85,B 0,C 180,E1 -3096.752,E2 -3096.752} C_VEL
LIN {X 0,Y 552.078,Z 866.526,A -85,B 0,C 180,E1 -3099.532,E2 -3099.532} C_VEL
LIN {X 0,Y 552.081,Z 866.526,A -85,B 0,C 180,E1 -3102.431,E2 -3102.431} C_VEL
LIN {X 0,Y 552.068,Z 866.525,A -85,B 0,C 180,E1 -3105.56,E2 -3105.56} C_VEL
LIN {X 0,Y 552.052,Z 866.532,A -85,B 0,C 180,E1 -3108.548,E2 -3108.548} C_VEL
LIN {X 0,Y 552.071,Z 866.523,A -85,B 0,C 180,E1 -3111.407,E2 -3111.407} C_VEL
LIN {X 0,Y 552.064,Z 866.534,A -85,B 0,C 180,E1 -3114.563,E2 -3114.563} C_VEL
LIN {X 0,Y 552.098,Z 866.523,A -85,B 0,C 180,E1 -3117.157,E2 -3117.157} C_VEL
LIN {X 0,Y 552.069,Z 866.523,A -85,B 0,C 180,E1 -3119.959,E2 -3119.959} C_VEL
LIN {X 0,Y 552.079,Z 866.531,A -85,B 0,C 180,E1 -3123.014,E2 -3123.014} C_VEL
LIN {X 0,Y 552.068,Z 866.523,A -85,B 0,C 180,E1 -3125.96,E2 -3125.96} C_VEL
LIN {X 0,Y 552.097,Z 866.529,A -85,B 0,C 180,E1 -3129.119,E2 -3129.119} C_VEL
LIN {X 0,Y 552.071,Z 866.531,A -85,B 0,C 180,E1 -3131.443,E2 -3131.443} C_VEL
LIN {X 0,Y 552.084,Z 866.526,A -85,B 0,C 180,E1 -3133.736,E2 -3133.736} C_VEL
LIN {X 0,Y 552.109,Z 866.521,A -85,B 0,C 180,E1 -3136.004,E2 -3136.004} C_VEL
LIN {X 0,Y 552.122,Z 866.517,A -85,B 0,C 180,E1 -3138.993,E2 -3138.993} C_VEL
LIN {X 0,Y 552.108,Z 866.526,A -85,B 0,C 180,E1 -3141.951,E2 -3141.951} C_VEL
LIN {X 0,Y 552.201,Z 866.506,A -85,B 0,C 180,E1 -3144.889,E2 -3144.889} C_VEL
LIN {X 0,Y 552.22,Z 866.511,A -85,B 0,C 180,E1 -3147.812,E2 -3147.812} C_VEL
LIN {X 0,Y 552.225,Z 866.512,A -85,B 0,C 180,E1 -3150,E2 -3150} C_VEL
LIN {X 0,Y 552.173,Z 866.511,A -85,B 0,C 180,E1 -3152.918,E2 -3152.918} C_VEL
LIN {X 0,Y 552.166,Z 866.513,A -85,B 0,C 180,E1 -3155.844,E2 -3155.844} C_VEL
LIN {X 0,Y 552.125,Z 866.522,A -85,B 0,C 180,E1 -3158.786,E2 -3158.786} C_VEL
LIN {X 0,Y 552.083,Z 866.521,A -85,B 0,C 180,E1 -3161.752,E2 -3161.752} C_VEL
LIN {X 0,Y 552.086,Z 866.529,A -85,B 0,C 180,E1 -3164.652,E2 -3164.652} C_VEL
LIN {X 0,Y 552.098,Z 866.523,A -85,B 0,C 180,E1 -3167.305,E2 -3167.305} C_VEL
LIN {X 0,Y 552.095,Z 866.52,A -85,B 0,C 180,E1 -3170.103,E2 -3170.103} C_VEL
LIN {X 0,Y 552.041,Z 866.527,A -85,B 0,C 180,E1 -3172.453,E2 -3172.453} C_VEL
LIN {X 0,Y 552.066,Z 866.533,A -85,B 0,C 180,E1 -3175.329,E2 -3175.329} C_VEL
LIN {X 0,Y 552.051,Z 866.526,A -85,B 0,C 180,E1 -3178.102,E2 -3178.102} C_VEL
LIN {X 0,Y 552.07,Z 866.523,A -85,B 0,C 180,E1 -3180.612,E2 -3180.612} C_VEL
LIN {X 0,Y 552.054,Z 866.529,A -85,B 0,C 180,E1 -3183.19,E2 -3183.19} C_VEL
LIN {X 0,Y 552.068,Z 866.532,A -85,B 0,C 180,E1 -3185.845,E2 -3185.845} C_VEL
LIN {X 0,Y 552.073,Z 866.523,A -85,B 0,C 180,E1 -3189.054,E2 -3189.054} C_VEL
LIN {X 0,Y 552.083,Z 866.525,A -85,B 0,C 180,E1 -3192.409,E2 -3192.409} C_VEL
LIN {X 0,Y 552.067,Z 866.525,A -85,B 0,C 180,E1 -3195.559,E2 -3195.559} C_VEL
LIN {X 0,Y 552.053,Z 866.531,A -85,B 0,C 180,E1 -3198.547,E2 -3198.547} C_VEL
LIN {X 0,Y 552.07,Z 866.523,A -85,B 0,C 180,E1 -3201.406,E2 -3201.406} C_VEL
LIN {X 0,Y 552.064,Z 866.534,A -85,B 0,C 180,E1 -3204.563,E2 -3204.563} C_VEL
LIN {X 0,Y 552.099,Z 866.522,A -85,B 0,C 180,E1 -3207.157,E2 -3207.157} C_VEL
LIN {X 0,Y 552.069,Z 866.523,A -85,B 0,C 180,E1 -3209.959,E2 -3209.959} C_VEL
LIN {X 0,Y 552.079,Z 866.531,A -85,B 0,C 180,E1 -3213.013,E2 -3213.013} C_VEL
LIN {X 0,Y 552.068,Z 866.523,A -85,B 0,C 180,E1 -3215.96,E2 -3215.96} C_VEL
LIN {X 0,Y 552.096,Z 866.529,A -85,B 0,C 180,E1 -3219.118,E2 -3219.118} C_VEL
LIN {X 0,Y 552.07,Z 866.531,A -85,B 0,C 180,E1 -3221.442,E2 -3221.442} C_VEL
LIN {X 0,Y 552.083,Z 866.526,A -85,B 0,C 180,E1 -3223.736,E2 -3223.736} C_VEL
LIN {X 0,Y 552.103,Z 866.521,A -85,B 0,C 180,E1 -3226.003,E2 -3226.003} C_VEL
LIN {X 0,Y 552.121,Z 866.518,A -85,B 0,C 180,E1 -3228.992,E2 -3228.992} C_VEL
LIN {X 0,Y 552.106,Z 866.526,A -85,B 0,C 180,E1 -3231.95,E2 -3231.95} C_VEL
LIN {X 0,Y 552.199,Z 866.507,A -85,B 0,C 180,E1 -3234.888,E2 -3234.888} C_VEL
LIN {X 0,Y 552.219,Z 866.511,A -85,B 0,C 180,E1 -3237.812,E2 -3237.812} C_VEL
LIN {X 0,Y 552.223,Z 866.512,A -85,B 0,C 180,E1 -3240,E2 -3240} C_VEL
LIN {X 0,Y 552.171,Z 866.511,A -85,B 0,C 180,E1 -3242.918,E2 -3242.918} C_VEL
LIN {X 0,Y 552.164,Z 866.513,A -85,B 0,C 180,E1 -3245.844,E2 -3245.844} C_VEL
LIN {X 0,Y 552.122,Z 866.522,A -85,B 0,C 180,E1 -3248.786,E2 -3248.786} C_VEL
LIN {X 0,Y 552.08,Z 866.522,A -85,B 0,C 180,E1 -3251.752,E2 -3251.752} C_VEL
LIN {X 0,Y 552.12,Z 866.527,A -85,B 0,C 180,E1 -3254.749,E2 -3254.749} C_VEL
LIN {X 0,Y 552.079,Z 866.522,A -85,B 0,C 180,E1 -3257.789,E2 -3257.789} C_VEL
LIN {X 0,Y 552.091,Z 866.52,A -85,B 0,C 180,E1 -3260.102,E2 -3260.102} C_VEL
LIN {X 0,Y 552.038,Z 866.528,A -85,B 0,C 180,E1 -3262.453,E2 -3262.453} C_VEL
LIN {X 0,Y 552.063,Z 866.533,A -85,B 0,C 180,E1 -3265.329,E2 -3265.329} C_VEL
LIN {X 0,Y 552.047,Z 866.526,A -85,B 0,C 180,E1 -3268.102,E2 -3268.102} C_VEL
LIN {X 0,Y 552.066,Z 866.523,A -85,B 0,C 180,E1 -3270.611,E2 -3270.611} C_VEL
LIN {X 0,Y 552.05,Z 866.529,A -85,B 0,C 180,E1 -3273.19,E2 -3273.19} C_VEL
LIN {X 0,Y 552.064,Z 866.532,A -85,B 0,C 180,E1 -3275.845,E2 -3275.845} C_VEL
LIN {X 0,Y 552.071,Z 866.523,A -85,B 0,C 180,E1 -3279.054,E2 -3279.054} C_VEL
LIN {X 0,Y 552.079,Z 866.526,A -85,B 0,C 180,E1 -3282.409,E2 -3282.409} C_VEL
LIN {X 0,Y 552.065,Z 866.525,A -85,B 0,C 180,E1 -3285.559,E2 -3285.559} C_VEL
LIN {X 0,Y 552.049,Z 866.531,A -85,B 0,C 180,E1 -3288.547,E2 -3288.547} C_VEL
LIN {X 0,Y 552.066,Z 866.523,A -85,B 0,C 180,E1 -3291.406,E2 -3291.406} C_VEL
LIN {X 0,Y 552.06,Z 866.534,A -85,B 0,C 180,E1 -3294.563,E2 -3294.563} C_VEL
LIN {X 0,Y 552.094,Z 866.522,A -85,B 0,C 180,E1 -3297.157,E2 -3297.157} C_VEL
LIN {X 0,Y 552.065,Z 866.524,A -85,B 0,C 180,E1 -3299.959,E2 -3299.959} C_VEL
LIN {X 0,Y 552.075,Z 866.533,A -85,B 0,C 180,E1 -3303.013,E2 -3303.013} C_VEL
LIN {X 0,Y 552.065,Z 866.527,A -85,B 0,C 180,E1 -3305.96,E2 -3305.96} C_VEL
LIN {X 0,Y 552.095,Z 866.666,A -85,B 0,C 180,E1 -3307.401,E2 -3307.401} C_VEL
LIN {X 0,Y 552.899,Z 871.97,A -85,B 0,C 180,E1 -3308.369,E2 -3308.369} C_VEL
LIN {X 0,Y 552.619,Z 887.602,A -85,B 0,C 180,E1 -3311.077,E2 -3311.077} C_VEL
LIN {X 0,Y 552.406,Z 903.234,A -85,B 0,C 180,E1 -3313.746,E2 -3313.746} C_VEL
LIN {X 0,Y 552.154,Z 921.099,A -85,B 0,C 180,E1 -3316.755,E2 -3316.755} C_VEL
LIN {X 0,Y 552.083,Z 932.723,A -85,B 0,C 180,E1 -3318.696,E2 -3318.696} C_VEL
LIN {X 0,Y 552.753,Z 940.071,A -85,B 0,C 180,E1 -3318.812,E2 -3318.812} C_VEL
LIN {X 0,Y 552.633,Z 1009.129,A -85,B 0,C 180,E1 -3319.721,E2 -3319.721} C_VEL
LIN {X 0,Y 552.497,Z 1018.406,A -85,B 0,C 180,E1 -3319.927,E2 -3319.927} C_VEL
LIN {X 0,Y 552.476,Z 1026.886,A -85,B 0,C 180,E1 -3320.204,E2 -3320.204} C_VEL
LIN {X 0,Y 552.385,Z 1035.395,A -85,B 0,C 180,E1 -3320.572,E2 -3320.572} C_VEL
LIN {X 0,Y 552.311,Z 1043.728,A -85,B 0,C 180,E1 -3321.032,E2 -3321.032} C_VEL
LIN {X 0,Y 552.162,Z 1051.767,A -85,B 0,C 180,E1 -3321.583,E2 -3321.583} C_VEL
LIN {X 0,Y 552.048,Z 1060.429,A -85,B 0,C 180,E1 -3322.318,E2 -3322.318} C_VEL
LIN {X 0,Y 551.953,Z 1069.431,A -85,B 0,C 180,E1 -3323.3,E2 -3323.3} C_VEL
LIN {X 0,Y 551.917,Z 1075.61,A -85,B 0,C 180,E1 -3324.153,E2 -3324.153} C_VEL
LIN {X 0,Y 551.746,Z 1079.987,A -85,B 0,C 180,E1 -3324.884,E2 -3324.884} C_VEL
LIN {X 0,Y 551.773,Z 1085.148,A -85,B 0,C 180,E1 -3325.983,E2 -3325.983} C_VEL
LIN {X 0,Y 551.766,Z 1087.788,A -85,B 0,C 180,E1 -3326.714,E2 -3326.714} C_VEL
LIN {X 0,Y 551.657,Z 1090.681,A -85,B 0,C 180,E1 -3327.81,E2 -3327.81} C_VEL
LIN {X 0,Y 551.643,Z 1091.934,A -85,B 0,C 180,E1 -3328.54,E2 -3328.54} C_VEL
LIN {X 0,Y 551.638,Z 1092.71,A -85,B 0,C 180,E1 -3329.27,E2 -3329.27} C_VEL
LIN {X 0,Y 551.637,Z 1093,A -85,B 0,C 180,E1 -3330,E2 -3330} C_VEL
LIN {X 0,Y 551.638,Z 1092.71,A -85,B 0,C 180,E1 -3330.73,E2 -3330.73} C_VEL
LIN {X 0,Y 551.643,Z 1091.935,A -85,B 0,C 180,E1 -3331.46,E2 -3331.46} C_VEL
LIN {X 0,Y 551.657,Z 1090.681,A -85,B 0,C 180,E1 -3332.19,E2 -3332.19} C_VEL
LIN {X 0,Y 551.761,Z 1087.788,A -85,B 0,C 180,E1 -3333.286,E2 -3333.286} C_VEL
LIN {X 0,Y 551.78,Z 1085.148,A -85,B 0,C 180,E1 -3334.017,E2 -3334.017} C_VEL
LIN {X 0,Y 551.745,Z 1079.986,A -85,B 0,C 180,E1 -3335.115,E2 -3335.115} C_VEL
LIN {X 0,Y 551.956,Z 1073.401,A -85,B 0,C 180,E1 -3336.184,E2 -3336.184} C_VEL
LIN {X 0,Y 551.992,Z 1065.745,A -85,B 0,C 180,E1 -3337.131,E2 -3337.131} C_VEL
LIN {X 0,Y 552.075,Z 1058.407,A -85,B 0,C 180,E1 -3337.865,E2 -3337.865} C_VEL
LIN {X 0,Y 552.197,Z 1050.546,A -85,B 0,C 180,E1 -3338.508,E2 -3338.508} C_VEL
LIN {X 0,Y 552.304,Z 1040.732,A -85,B 0,C 180,E1 -3339.152,E2 -3339.152} C_VEL
LIN {X 0,Y 552.451,Z 1029.305,A -85,B 0,C 180,E1 -3339.704,E2 -3339.704} C_VEL
LIN {X 0,Y 552.511,Z 1019.25,A -85,B 0,C 180,E1 -3340.05,E2 -3340.05} C_VEL
LIN {X 0,Y 552.577,Z 1010.448,A -85,B 0,C 180,E1 -3340.257,E2 -3340.257} C_VEL
LIN {X 0,Y 552.742,Z 969.291,A -85,B 0,C 180,E1 -3340.809,E2 -3340.809} C_VEL
LIN {X 0,Y 552.612,Z 937.019,A -85,B 0,C 180,E1 -3341.23,E2 -3341.23} C_VEL
LIN {X 0,Y 552.063,Z 932.72,A -85,B 0,C 180,E1 -3341.305,E2 -3341.305} C_VEL
LIN {X 0,Y 552.208,Z 915.545,A -85,B 0,C 180,E1 -3344.177,E2 -3344.177} C_VEL
LIN {X 0,Y 552.476,Z 898.77,A -85,B 0,C 180,E1 -3347.012,E2 -3347.012} C_VEL
LIN {X 0,Y 552.773,Z 880.904,A -85,B 0,C 180,E1 -3350.077,E2 -3350.077} C_VEL
LIN {X 0,Y 552.778,Z 870.712,A -85,B 0,C 180,E1 -3351.857,E2 -3351.857} C_VEL
LIN {X 0,Y 552.08,Z 866.532,A -85,B 0,C 180,E1 -3352.649,E2 -3352.649} C_VEL
LIN {X 0,Y 552.046,Z 866.53,A -85,B 0,C 180,E1 -3355.648,E2 -3355.648} C_VEL
LIN {X 0,Y 552.068,Z 866.526,A -85,B 0,C 180,E1 -3358.551,E2 -3358.551} C_VEL
LIN {X 0,Y 552.09,Z 866.529,A -85,B 0,C 180,E1 -3361.472,E2 -3361.472} C_VEL
LIN {X 0,Y 552.091,Z 866.522,A -85,B 0,C 180,E1 -3364.164,E2 -3364.164} C_VEL
LIN {X 0,Y 552.041,Z 866.527,A -85,B 0,C 180,E1 -3366.752,E2 -3366.752} C_VEL
LIN {X 0,Y 552.067,Z 866.533,A -85,B 0,C 180,E1 -3369.533,E2 -3369.533} C_VEL
LIN {X 0,Y 552.076,Z 866.524,A -85,B 0,C 180,E1 -3372.431,E2 -3372.431} C_VEL
LIN {X 0,Y 552.062,Z 866.529,A -85,B 0,C 180,E1 -3375.559,E2 -3375.559} C_VEL
LIN {X 0,Y 552.048,Z 866.529,A -85,B 0,C 180,E1 -3378.548,E2 -3378.548} C_VEL
LIN {X 0,Y 552.067,Z 866.524,A -85,B 0,C 180,E1 -3381.407,E2 -3381.407} C_VEL
LIN {X 0,Y 552.058,Z 866.531,A -85,B 0,C 180,E1 -3384.563,E2 -3384.563} C_VEL
LIN {X 0,Y 552.093,Z 866.522,A -85,B 0,C 180,E1 -3387.157,E2 -3387.157} C_VEL
LIN {X 0,Y 552.064,Z 866.526,A -85,B 0,C 180,E1 -3389.959,E2 -3389.959} C_VEL
LIN {X 0,Y 552.073,Z 866.529,A -85,B 0,C 180,E1 -3393.014,E2 -3393.014} C_VEL
LIN {X 0,Y 552.058,Z 866.527,A -85,B 0,C 180,E1 -3395.96,E2 -3395.96} C_VEL
LIN {X 0,Y 552.07,Z 866.533,A -85,B 0,C 180,E1 -3399.118,E2 -3399.118} C_VEL
LIN {X 0,Y 552.069,Z 866.532,A -85,B 0,C 180,E1 -3401.443,E2 -3401.443} C_VEL
LIN {X 0,Y 552.132,Z 866.673,A -85,B 0,C 180,E1 -3402.46,E2 -3402.46} C_VEL
LIN {X 0,Y 552.041,Z 878.957,A -85,B 0,C 180,E1 -3405.249,E2 -3405.249} C_VEL
LIN {X 0,Y 551.929,Z 892.322,A -85,B 0,C 180,E1 -3408.245,E2 -3408.245} C_VEL
LIN {X 0,Y 551.908,Z 894.629,A -85,B 0,C 180,E1 -3408.758,E2 -3408.758} C_VEL
LIN {X 0,Y 552.785,Z 902.281,A -85,B 0,C 180,E1 -3408.886,E2 -3408.886} C_VEL
LIN {X 0,Y 552.597,Z 969.236,A -85,B 0,C 180,E1 -3409.767,E2 -3409.767} C_VEL
LIN {X 0,Y 552.548,Z 978.481,A -85,B 0,C 180,E1 -3409.974,E2 -3409.974} C_VEL
LIN {X 0,Y 552.432,Z 988.152,A -85,B 0,C 180,E1 -3410.296,E2 -3410.296} C_VEL
LIN {X 0,Y 552.352,Z 998.23,A -85,B 0,C 180,E1 -3410.756,E2 -3410.756} C_VEL
LIN {X 0,Y 552.23,Z 1008.729,A -85,B 0,C 180,E1 -3411.4,E2 -3411.4} C_VEL
LIN {X 0,Y 552.077,Z 1017.945,A -85,B 0,C 180,E1 -3412.135,E2 -3412.135} C_VEL
LIN {X 0,Y 552.004,Z 1025.378,A -85,B 0,C 180,E1 -3412.87,E2 -3412.87} C_VEL
LIN {X 0,Y 551.932,Z 1033.053,A -85,B 0,C 180,E1 -3413.816,E2 -3413.816} C_VEL
LIN {X 0,Y 551.746,Z 1039.77,A -85,B 0,C 180,E1 -3414.885,E2 -3414.885} C_VEL
LIN {X 0,Y 551.78,Z 1045.008,A -85,B 0,C 180,E1 -3415.983,E2 -3415.983} C_VEL
LIN {X 0,Y 551.73,Z 1048.804,A -85,B 0,C 180,E1 -3417.08,E2 -3417.08} C_VEL
LIN {X 0,Y 551.657,Z 1050.613,A -85,B 0,C 180,E1 -3417.81,E2 -3417.81} C_VEL
LIN {X 0,Y 551.643,Z 1051.915,A -85,B 0,C 180,E1 -3418.54,E2 -3418.54} C_VEL
LIN {X 0,Y 551.638,Z 1052.715,A -85,B 0,C 180,E1 -3419.27,E2 -3419.27} C_VEL
LIN {X 0,Y 551.638,Z 1052.996,A -85,B 0,C 180,E1 -3420,E2 -3420} C_VEL
LIN {X 0,Y 551.639,Z 1052.76,A -85,B 0,C 180,E1 -3420.73,E2 -3420.73} C_VEL
LIN {X 0,Y 551.645,Z 1052.03,A -85,B 0,C 180,E1 -3421.46,E2 -3421.46} C_VEL
LIN {X 0,Y 551.658,Z 1050.809,A -85,B 0,C 180,E1 -3422.191,E2 -3422.191} C_VEL
LIN {X 0,Y 551.761,Z 1047.957,A -85,B 0,C 180,E1 -3423.286,E2 -3423.286} C_VEL
LIN {X 0,Y 551.806,Z 1043.852,A -85,B 0,C 180,E1 -3424.383,E2 -3424.383} C_VEL
LIN {X 0,Y 551.82,Z 1038.239,A -85,B 0,C 180,E1 -3425.482,E2 -3425.482} C_VEL
LIN {X 0,Y 551.926,Z 1031.878,A -85,B 0,C 180,E1 -3426.436,E2 -3426.436} C_VEL
LIN {X 0,Y 551.996,Z 1024.502,A -85,B 0,C 180,E1 -3427.315,E2 -3427.315} C_VEL
LIN {X 0,Y 552.104,Z 1015.866,A -85,B 0,C 180,E1 -3428.142,E2 -3428.142} C_VEL
LIN {X 0,Y 552.302,Z 1005.996,A -85,B 0,C 180,E1 -3428.876,E2 -3428.876} C_VEL
LIN {X 0,Y 552.359,Z 996.316,A -85,B 0,C 180,E1 -3429.429,E2 -3429.429} C_VEL
LIN {X 0,Y 552.449,Z 988.07,A -85,B 0,C 180,E1 -3429.797,E2 -3429.797} C_VEL
LIN {X 0,Y 552.525,Z 978.364,A -85,B 0,C 180,E1 -3430.119,E2 -3430.119} C_VEL
LIN {X 0,Y 552.627,Z 969.053,A -85,B 0,C 180,E1 -3430.326,E2 -3430.326} C_VEL
LIN {X 0,Y 552.636,Z 899.555,A -85,B 0,C 180,E1 -3431.242,E2 -3431.242} C_VEL
LIN {X 0,Y 551.94,Z 894.569,A -85,B 0,C 180,E1 -3431.344,E2 -3431.344} C_VEL
LIN {X 0,Y 552.004,Z 881.304,A -85,B 0,C 180,E1 -3434.313,E2 -3434.313} C_VEL
LIN {X 0,Y 552.204,Z 867.919,A -85,B 0,C 180,E1 -3437.343,E2 -3437.343} C_VEL
LIN {X 0,Y 552.135,Z 866.519,A -85,B 0,C 180,E1 -3437.719,E2 -3437.719} C_VEL
LIN {X 0,Y 552.092,Z 866.52,A -85,B 0,C 180,E1 -3440.103,E2 -3440.103} C_VEL
LIN {X 0,Y 552.039,Z 866.528,A -85,B 0,C 180,E1 -3442.454,E2 -3442.454} C_VEL
LIN {X 0,Y 552.039,Z 866.535,A -85,B 0,C 180,E1 -3443.161,E2 -3443.161} C_VEL
LIN {X 0,Y 551.403,Z 866.62,A -85,B 0,C 180,E1 -3443.771,E2 -3443.771} C_VEL
LIN {X 0,Y 548.559,Z 866.972,A -85,B 0,C 180,E1 -3444.76,E2 -3444.76} C_VEL
LIN {X 0,Y 546.139,Z 867.268,A -85,B 0,C 180,E1 -3445.556,E2 -3445.556} C_VEL
LIN {X 0,Y 545.105,Z 867.391,A -85,B 0,C 180,E1 -3446.171,E2 -3446.171} C_VEL
LIN {X 0,Y 545.024,Z 867.401,A -85,B 0,C 180,E1 -3446.379,E2 -3446.379} C_VEL
LIN {X 0,Y 545.012,Z 867.411,A -85,B 0,C 180,E1 -3449.342,E2 -3449.342} C_VEL
LIN {X 0,Y 545.041,Z 867.403,A -85,B 0,C 180,E1 -3451.916,E2 -3451.916} C_VEL
LIN {X 0,Y 545.046,Z 867.398,A -85,B 0,C 180,E1 -3454.566,E2 -3454.566} C_VEL
LIN {X 0,Y 545.008,Z 867.405,A -85,B 0,C 180,E1 -3457.307,E2 -3457.307} C_VEL
LIN {X 0,Y 545.008,Z 867.409,A -85,B 0,C 180,E1 -3460.148,E2 -3460.148} C_VEL
LIN {X 0,Y 545.018,Z 867.401,A -85,B 0,C 180,E1 -3463.113,E2 -3463.113} C_VEL
LIN {X 0,Y 545.026,Z 867.41,A -85,B 0,C 180,E1 -3466.23,E2 -3466.23} C_VEL
LIN {X 0,Y 544.995,Z 867.406,A -85,B 0,C 180,E1 -3468.877,E2 -3468.877} C_VEL
LIN {X 0,Y 545.021,Z 867.403,A -85,B 0,C 180,E1 -3471.869,E2 -3471.869} C_VEL
LIN {X 0,Y 545.024,Z 867.411,A -85,B 0,C 180,E1 -3474.531,E2 -3474.531} C_VEL
LIN {X 0,Y 545.053,Z 867.4,A -85,B 0,C 180,E1 -3477.211,E2 -3477.211} C_VEL
LIN {X 0,Y 545.019,Z 867.401,A -85,B 0,C 180,E1 -3479.808,E2 -3479.808} C_VEL
LIN {X 0,Y 545,Z 867.406,A -85,B 0,C 180,E1 -3482.339,E2 -3482.339} C_VEL
LIN {X 0,Y 545.023,Z 867.408,A -85,B 0,C 180,E1 -3484.816,E2 -3484.816} C_VEL
LIN {X 0,Y 545.01,Z 867.411,A -85,B 0,C 180,E1 -3487.241,E2 -3487.241} C_VEL
LIN {X 0,Y 545.092,Z 867.392,A -85,B 0,C 180,E1 -3490.257,E2 -3490.257} C_VEL
LIN {X 0,Y 545.054,Z 867.398,A -85,B 0,C 180,E1 -3492.749,E2 -3492.749} C_VEL
LIN {X 0,Y 545.069,Z 867.4,A -85,B 0,C 180,E1 -3495.819,E2 -3495.819} C_VEL
LIN {X 0,Y 545.07,Z 867.395,A -85,B 0,C 180,E1 -3498.848,E2 -3498.848} C_VEL
LIN {X 0,Y 545.066,Z 867.405,A -85,B 0,C 180,E1 -3501.846,E2 -3501.846} C_VEL
LIN {X 0,Y 545.159,Z 867.384,A -85,B 0,C 180,E1 -3504.823,E2 -3504.823} C_VEL
LIN {X 0,Y 545.191,Z 867.386,A -85,B 0,C 180,E1 -3507.784,E2 -3507.784} C_VEL
LIN {X 0,Y 545.193,Z 867.388,A -85,B 0,C 180,E1 -3510,E2 -3510} C_VEL
LIN {X 0,Y 545.141,Z 867.387,A -85,B 0,C 180,E1 -3512.956,E2 -3512.956} C_VEL
LIN {X 0,Y 545.119,Z 867.392,A -85,B 0,C 180,E1 -3515.92,E2 -3515.92} C_VEL
LIN {X 0,Y 545.068,Z 867.4,A -85,B 0,C 180,E1 -3518.901,E2 -3518.901} C_VEL
LIN {X 0,Y 545.056,Z 867.397,A -85,B 0,C 180,E1 -3521.906,E2 -3521.906} C_VEL
LIN {X 0,Y 545.04,Z 867.407,A -85,B 0,C 180,E1 -3524.945,E2 -3524.945} C_VEL
LIN {X 0,Y 545.049,Z 867.398,A -85,B 0,C 180,E1 -3528.027,E2 -3528.027} C_VEL
LIN {X 0,Y 545.033,Z 867.401,A -85,B 0,C 180,E1 -3530.375,E2 -3530.375} C_VEL
LIN {X 0,Y 544.988,Z 867.409,A -85,B 0,C 180,E1 -3532.76,E2 -3532.76} C_VEL
LIN {X 0,Y 545.013,Z 867.409,A -85,B 0,C 180,E1 -3535.489,E2 -3535.489} C_VEL
LIN {X 0,Y 545.001,Z 867.409,A -85,B 0,C 180,E1 -3537.661,E2 -3537.661} C_VEL
LIN {X 0,Y 545.024,Z 867.401,A -85,B 0,C 180,E1 -3540.235,E2 -3540.235} C_VEL
LIN {X 0,Y 545.032,Z 867.402,A -85,B 0,C 180,E1 -3543.054,E2 -3543.054} C_VEL
LIN {X 0,Y 545.019,Z 867.411,A -85,B 0,C 180,E1 -3545.67,E2 -3545.67} C_VEL
LIN {X 0,Y 545.018,Z 867.405,A -85,B 0,C 180,E1 -3548.241,E2 -3548.241} C_VEL
LIN {X 0,Y 544.997,Z 867.404,A -85,B 0,C 180,E1 -3551.123,E2 -3551.123} C_VEL
LIN {X 0,Y 545.028,Z 867.41,A -85,B 0,C 180,E1 -3554.133,E2 -3554.133} C_VEL
LIN {X 0,Y 545.002,Z 867.405,A -85,B 0,C 180,E1 -3556.885,E2 -3556.885} C_VEL
LIN {X 0,Y 545.008,Z 867.405,A -85,B 0,C 180,E1 -3559.852,E2 -3559.852} C_VEL
LIN {X 0,Y 544.994,Z 867.411,A -85,B 0,C 180,E1 -3562.692,E2 -3562.692} C_VEL
LIN {X 0,Y 545.055,Z 867.397,A -85,B 0,C 180,E1 -3565.612,E2 -3565.612} C_VEL
LIN {X 0,Y 545.046,Z 867.402,A -85,B 0,C 180,E1 -3568.324,E2 -3568.324} C_VEL
LIN {X 0,Y 545.034,Z 867.401,A -85,B 0,C 180,E1 -3571.503,E2 -3571.503} C_VEL
LIN {X 0,Y 545.02,Z 867.401,A -85,B 0,C 180,E1 -3573.996,E2 -3573.996} C_VEL
LIN {X 0,Y 545.071,Z 867.396,A -85,B 0,C 180,E1 -3576.44,E2 -3576.44} C_VEL
LIN {X 0,Y 545.036,Z 867.404,A -85,B 0,C 180,E1 -3578.835,E2 -3578.835} C_VEL
LIN {X 0,Y 545.032,Z 867.409,A -85,B 0,C 180,E1 -3581.193,E2 -3581.193} C_VEL
LIN {X 0,Y 545.036,Z 867.407,A -85,B 0,C 180,E1 -3583.52,E2 -3583.52} C_VEL
LIN {X 0,Y 545.064,Z 867.401,A -85,B 0,C 180,E1 -3585.819,E2 -3585.819} C_VEL
LIN {X 0,Y 545.069,Z 867.395,A -85,B 0,C 180,E1 -3588.848,E2 -3588.848} C_VEL
LIN {X 0,Y 545.064,Z 867.405,A -85,B 0,C 180,E1 -3591.846,E2 -3591.846} C_VEL
LIN {X 0,Y 545.157,Z 867.384,A -85,B 0,C 180,E1 -3594.822,E2 -3594.822} C_VEL
LIN {X 0,Y 545.19,Z 867.386,A -85,B 0,C 180,E1 -3597.783,E2 -3597.783} C_VEL
LIN {X 0,Y 545.191,Z 867.388,A -85,B 0,C 180,E1 -3600,E2 -3600} C_VEL
LIN {X 0,Y 545.138,Z 867.387,A -85,B 0,C 180,E1 -3602.956,E2 -3602.956} C_VEL
LIN {X 0,Y 545.116,Z 867.392,A -85,B 0,C 180,E1 -3605.92,E2 -3605.92} C_VEL
LIN {X 0,Y 545.065,Z 867.4,A -85,B 0,C 180,E1 -3608.901,E2 -3608.901} C_VEL
LIN {X 0,Y 545.053,Z 867.398,A -85,B 0,C 180,E1 -3611.906,E2 -3611.906} C_VEL
LIN {X 0,Y 545.054,Z 867.404,A -85,B 0,C 180,E1 -3614.944,E2 -3614.944} C_VEL
LIN {X 0,Y 545.046,Z 867.398,A -85,B 0,C 180,E1 -3618.027,E2 -3618.027} C_VEL
LIN {X 0,Y 545.03,Z 867.401,A -85,B 0,C 180,E1 -3620.374,E2 -3620.374} C_VEL
LIN {X 0,Y 544.985,Z 867.41,A -85,B 0,C 180,E1 -3622.76,E2 -3622.76} C_VEL
LIN {X 0,Y 545.009,Z 867.409,A -85,B 0,C 180,E1 -3625.489,E2 -3625.489} C_VEL
LIN {X 0,Y 544.997,Z 867.409,A -85,B 0,C 180,E1 -3627.661,E2 -3627.661} C_VEL
LIN {X 0,Y 545.02,Z 867.402,A -85,B 0,C 180,E1 -3630.235,E2 -3630.235} C_VEL
LIN {X 0,Y 545.028,Z 867.402,A -85,B 0,C 180,E1 -3633.053,E2 -3633.053} C_VEL
LIN {X 0,Y 545.016,Z 867.412,A -85,B 0,C 180,E1 -3635.67,E2 -3635.67} C_VEL
LIN {X 0,Y 545.016,Z 867.405,A -85,B 0,C 180,E1 -3638.24,E2 -3638.24} C_VEL
LIN {X 0,Y 544.993,Z 867.405,A -85,B 0,C 180,E1 -3641.122,E2 -3641.122} C_VEL
LIN {X 0,Y 545.028,Z 867.41,A -85,B 0,C 180,E1 -3644.132,E2 -3644.132} C_VEL
LIN {X 0,Y 544.997,Z 867.405,A -85,B 0,C 180,E1 -3646.885,E2 -3646.885} C_VEL
LIN {X 0,Y 545.004,Z 867.406,A -85,B 0,C 180,E1 -3649.852,E2 -3649.852} C_VEL
LIN {X 0,Y 544.99,Z 867.411,A -85,B 0,C 180,E1 -3652.692,E2 -3652.692} C_VEL
LIN {X 0,Y 545.051,Z 867.397,A -85,B 0,C 180,E1 -3655.612,E2 -3655.612} C_VEL
LIN {X 0,Y 545.042,Z 867.403,A -85,B 0,C 180,E1 -3658.324,E2 -3658.324} C_VEL
LIN {X 0,Y 545.03,Z 867.401,A -85,B 0,C 180,E1 -3661.503,E2 -3661.503} C_VEL
LIN {X 0,Y 545.016,Z 867.404,A -85,B 0,C 180,E1 -3663.996,E2 -3663.996} C_VEL
LIN {X 0,Y 545.06,Z 867.504,A -85,B 0,C 180,E1 -3667.243,E2 -3667.243} C_VEL
LIN {X 0,Y 545.94,Z 873.087,A -85,B 0,C 180,E1 -3668.278,E2 -3668.278} C_VEL
LIN {X 0,Y 545.649,Z 888.719,A -85,B 0,C 180,E1 -3671.021,E2 -3671.021} C_VEL
LIN {X 0,Y 545.345,Z 905.467,A -85,B 0,C 180,E1 -3673.914,E2 -3673.914} C_VEL
LIN {X 0,Y 545.109,Z 922.216,A -85,B 0,C 180,E1 -3676.771,E2 -3676.771} C_VEL
LIN {X 0,Y 545.044,Z 932.755,A -85,B 0,C 180,E1 -3678.554,E2 -3678.554} C_VEL
LIN {X 0,Y 545.788,Z 940.185,A -85,B 0,C 180,E1 -3678.669,E2 -3678.669} C_VEL
LIN {X 0,Y 545.669,Z 1009.129,A -85,B 0,C 180,E1 -3679.588,E2 -3679.588} C_VEL
LIN {X 0,Y 545.516,Z 1018.406,A -85,B 0,C 180,E1 -3679.796,E2 -3679.796} C_VEL
LIN {X 0,Y 545.497,Z 1026.884,A -85,B 0,C 180,E1 -3680.077,E2 -3680.077} C_VEL
LIN {X 0,Y 545.392,Z 1035.393,A -85,B 0,C 180,E1 -3680.45,E2 -3680.45} C_VEL
LIN {X 0,Y 545.276,Z 1043.726,A -85,B 0,C 180,E1 -3680.915,E2 -3680.915} C_VEL
LIN {X 0,Y 545.141,Z 1051.767,A -85,B 0,C 180,E1 -3681.474,E2 -3681.474} C_VEL
LIN {X 0,Y 545.008,Z 1060.429,A -85,B 0,C 180,E1 -3682.218,E2 -3682.218} C_VEL
LIN {X 0,Y 544.903,Z 1069.08,A -85,B 0,C 180,E1 -3683.167,E2 -3683.167} C_VEL
LIN {X 0,Y 544.843,Z 1075.61,A -85,B 0,C 180,E1 -3684.077,E2 -3684.077} C_VEL
LIN {X 0,Y 544.672,Z 1079.987,A -85,B 0,C 180,E1 -3684.818,E2 -3684.818} C_VEL
LIN {X 0,Y 544.697,Z 1085.148,A -85,B 0,C 180,E1 -3685.93,E2 -3685.93} C_VEL
LIN {X 0,Y 544.659,Z 1088.935,A -85,B 0,C 180,E1 -3687.041,E2 -3687.041} C_VEL
LIN {X 0,Y 544.571,Z 1090.682,A -85,B 0,C 180,E1 -3687.781,E2 -3687.781} C_VEL
LIN {X 0,Y 544.544,Z 1091.934,A -85,B 0,C 180,E1 -3688.521,E2 -3688.521} C_VEL
LIN {X 0,Y 544.538,Z 1092.709,A -85,B 0,C 180,E1 -3689.26,E2 -3689.26} C_VEL
LIN {X 0,Y 544.538,Z 1093,A -85,B 0,C 180,E1 -3690,E2 -3690} C_VEL
LIN {X 0,Y 544.538,Z 1092.709,A -85,B 0,C 180,E1 -3690.739,E2 -3690.739} C_VEL
LIN {X 0,Y 544.544,Z 1091.934,A -85,B 0,C 180,E1 -3691.479,E2 -3691.479} C_VEL
LIN {X 0,Y 544.571,Z 1090.682,A -85,B 0,C 180,E1 -3692.219,E2 -3692.219} C_VEL
LIN {X 0,Y 544.688,Z 1087.788,A -85,B 0,C 180,E1 -3693.328,E2 -3693.328} C_VEL
LIN {X 0,Y 544.703,Z 1085.149,A -85,B 0,C 180,E1 -3694.069,E2 -3694.069} C_VEL
LIN {X 0,Y 544.672,Z 1079.986,A -85,B 0,C 180,E1 -3695.182,E2 -3695.182} C_VEL
LIN {X 0,Y 544.88,Z 1073.957,A -85,B 0,C 180,E1 -3696.183,E2 -3696.183} C_VEL
LIN {X 0,Y 544.92,Z 1065.745,A -85,B 0,C 180,E1 -3697.224,E2 -3697.224} C_VEL
LIN {X 0,Y 545.034,Z 1058.406,A -85,B 0,C 180,E1 -3697.968,E2 -3697.968} C_VEL
LIN {X 0,Y 545.164,Z 1050.544,A -85,B 0,C 180,E1 -3698.619,E2 -3698.619} C_VEL
LIN {X 0,Y 545.266,Z 1042.231,A -85,B 0,C 180,E1 -3699.178,E2 -3699.178} C_VEL
LIN {X 0,Y 545.425,Z 1031.615,A -85,B 0,C 180,E1 -3699.737,E2 -3699.737} C_VEL
LIN {X 0,Y 545.54,Z 1020.08,A -85,B 0,C 180,E1 -3700.156,E2 -3700.156} C_VEL
LIN {X 0,Y 545.612,Z 1010.447,A -85,B 0,C 180,E1 -3700.389,E2 -3700.389} C_VEL
LIN {X 0,Y 545.784,Z 956.77,A -85,B 0,C 180,E1 -3701.113,E2 -3701.113} C_VEL
LIN {X 0,Y 545.699,Z 937.901,A -85,B 0,C 180,E1 -3701.363,E2 -3701.363} C_VEL
LIN {X 0,Y 544.972,Z 932.745,A -85,B 0,C 180,E1 -3701.45,E2 -3701.45} C_VEL
LIN {X 0,Y 545.201,Z 916.635,A -85,B 0,C 180,E1 -3704.177,E2 -3704.177} C_VEL
LIN {X 0,Y 545.477,Z 898.77,A -85,B 0,C 180,E1 -3707.238,E2 -3707.238} C_VEL
LIN {X 0,Y 545.799,Z 882.393,A -85,B 0,C 180,E1 -3710.083,E2 -3710.083} C_VEL
LIN {X 0,Y 545.777,Z 871.532,A -85,B 0,C 180,E1 -3712.006,E2 -3712.006} C_VEL
LIN {X 0,Y 545.046,Z 867.408,A -85,B 0,C 180,E1 -3712.807,E2 -3712.807} C_VEL
LIN {X 0,Y 545.015,Z 867.405,A -85,B 0,C 180,E1 -3716.004,E2 -3716.004} C_VEL
LIN {X 0,Y 545.014,Z 867.407,A -85,B 0,C 180,E1 -3718.734,E2 -3718.734} C_VEL
LIN {X 0,Y 545.04,Z 867.405,A -85,B 0,C 180,E1 -3721.676,E2 -3721.676} C_VEL
LIN {X 0,Y 545.042,Z 867.4,A -85,B 0,C 180,E1 -3724.566,E2 -3724.566} C_VEL
LIN {X 0,Y 544.989,Z 867.412,A -85,B 0,C 180,E1 -3727.308,E2 -3727.308} C_VEL
LIN {X 0,Y 545.002,Z 867.407,A -85,B 0,C 180,E1 -3730.148,E2 -3730.148} C_VEL
LIN {X 0,Y 544.996,Z 867.406,A -85,B 0,C 180,E1 -3733.115,E2 -3733.115} C_VEL
LIN {X 0,Y 545.021,Z 867.407,A -85,B 0,C 180,E1 -3736.229,E2 -3736.229} C_VEL
LIN {X 0,Y 544.991,Z 867.406,A -85,B 0,C 180,E1 -3738.877,E2 -3738.877} C_VEL
LIN {X 0,Y 545.013,Z 867.407,A -85,B 0,C 180,E1 -3741.869,E2 -3741.869} C_VEL
LIN {X 0,Y 545.018,Z 867.409,A -85,B 0,C 180,E1 -3744.53,E2 -3744.53} C_VEL
LIN {X 0,Y 545.048,Z 867.399,A -85,B 0,C 180,E1 -3747.21,E2 -3747.21} C_VEL
LIN {X 0,Y 545.014,Z 867.403,A -85,B 0,C 180,E1 -3749.808,E2 -3749.808} C_VEL
LIN {X 0,Y 544.994,Z 867.41,A -85,B 0,C 180,E1 -3752.339,E2 -3752.339} C_VEL
LIN {X 0,Y 545.017,Z 867.413,A -85,B 0,C 180,E1 -3754.816,E2 -3754.816} C_VEL
LIN {X 0,Y 544.982,Z 867.414,A -85,B 0,C 180,E1 -3757.24,E2 -3757.24} C_VEL
LIN {X 0,Y 545.057,Z 867.399,A -85,B 0,C 180,E1 -3760.266,E2 -3760.266} C_VEL
LIN {X 0,Y 545.077,Z 867.484,A -85,B 0,C 180,E1 -3762.413,E2 -3762.413} C_VEL
LIN {X 0,Y 545.007,Z 878.96,A -85,B 0,C 180,E1 -3765.054,E2 -3765.054} C_VEL
LIN {X 0,Y 544.879,Z 892.325,A -85,B 0,C 180,E1 -3768.09,E2 -3768.09} C_VEL
LIN {X 0,Y 544.868,Z 894.644,A -85,B 0,C 180,E1 -3768.614,E2 -3768.614} C_VEL
LIN {X 0,Y 545.816,Z 901.382,A -85,B 0,C 180,E1 -3768.73,E2 -3768.73} C_VEL
LIN {X 0,Y 545.614,Z 969.269,A -85,B 0,C 180,E1 -3769.635,E2 -3769.635} C_VEL
LIN {X 0,Y 545.548,Z 978.501,A -85,B 0,C 180,E1 -3769.844,E2 -3769.844} C_VEL
LIN {X 0,Y 545.446,Z 988.17,A -85,B 0,C 180,E1 -3770.17,E2 -3770.17} C_VEL
LIN {X 0,Y 545.34,Z 998.245,A -85,B 0,C 180,E1 -3770.636,E2 -3770.636} C_VEL
LIN {X 0,Y 545.223,Z 1008.732,A -85,B 0,C 180,E1 -3771.289,E2 -3771.289} C_VEL
LIN {X 0,Y 545.038,Z 1017.956,A -85,B 0,C 180,E1 -3772.033,E2 -3772.033} C_VEL
LIN {X 0,Y 544.948,Z 1025.389,A -85,B 0,C 180,E1 -3772.777,E2 -3772.777} C_VEL
LIN {X 0,Y 544.863,Z 1031.755,A -85,B 0,C 180,E1 -3773.554,E2 -3773.554} C_VEL
LIN {X 0,Y 544.711,Z 1038.785,A -85,B 0,C 180,E1 -3774.633,E2 -3774.633} C_VEL
LIN {X 0,Y 544.711,Z 1043.445,A -85,B 0,C 180,E1 -3775.56,E2 -3775.56} C_VEL
LIN {X 0,Y 544.689,Z 1047.682,A -85,B 0,C 180,E1 -3776.672,E2 -3776.672} C_VEL
LIN {X 0,Y 544.572,Z 1050.618,A -85,B 0,C 180,E1 -3777.781,E2 -3777.781} C_VEL
LIN {X 0,Y 544.544,Z 1051.92,A -85,B 0,C 180,E1 -3778.521,E2 -3778.521} C_VEL
LIN {X 0,Y 544.538,Z 1052.717,A -85,B 0,C 180,E1 -3779.261,E2 -3779.261} C_VEL
LIN {X 0,Y 544.539,Z 1052.996,A -85,B 0,C 180,E1 -3780,E2 -3780} C_VEL
LIN {X 0,Y 544.539,Z 1052.763,A -85,B 0,C 180,E1 -3780.74,E2 -3780.74} C_VEL
LIN {X 0,Y 544.545,Z 1052.034,A -85,B 0,C 180,E1 -3781.479,E2 -3781.479} C_VEL
LIN {X 0,Y 544.573,Z 1050.812,A -85,B 0,C 180,E1 -3782.219,E2 -3782.219} C_VEL
LIN {X 0,Y 544.688,Z 1047.959,A -85,B 0,C 180,E1 -3783.329,E2 -3783.329} C_VEL
LIN {X 0,Y 544.707,Z 1043.847,A -85,B 0,C 180,E1 -3784.44,E2 -3784.44} C_VEL
LIN {X 0,Y 544.763,Z 1038.235,A -85,B 0,C 180,E1 -3785.553,E2 -3785.553} C_VEL
LIN {X 0,Y 544.848,Z 1031.497,A -85,B 0,C 180,E1 -3786.568,E2 -3786.568} C_VEL
LIN {X 0,Y 544.931,Z 1024.501,A -85,B 0,C 180,E1 -3787.41,E2 -3787.41} C_VEL
LIN {X 0,Y 545.087,Z 1015.859,A -85,B 0,C 180,E1 -3788.247,E2 -3788.247} C_VEL
LIN {X 0,Y 545.29,Z 1005.991,A -85,B 0,C 180,E1 -3788.991,E2 -3788.991} C_VEL
LIN {X 0,Y 545.36,Z 996.308,A -85,B 0,C 180,E1 -3789.551,E2 -3789.551} C_VEL
LIN {X 0,Y 545.458,Z 986.84,A -85,B 0,C 180,E1 -3789.971,E2 -3789.971} C_VEL
LIN {X 0,Y 545.559,Z 976.669,A -85,B 0,C 180,E1 -3790.297,E2 -3790.297} C_VEL
LIN {X 0,Y 545.681,Z 964.882,A -85,B 0,C 180,E1 -3790.529,E2 -3790.529} C_VEL
LIN {X 0,Y 545.72,Z 900.596,A -85,B 0,C 180,E1 -3791.372,E2 -3791.372} C_VEL
LIN {X 0,Y 544.875,Z 894.604,A -85,B 0,C 180,E1 -3791.485,E2 -3791.485} C_VEL
LIN {X 0,Y 544.948,Z 881.535,A -85,B 0,C 180,E1 -3794.449,E2 -3794.449} C_VEL
LIN {X 0,Y 545.177,Z 868.426,A -85,B 0,C 180,E1 -3797.455,E2 -3797.455} C_VEL
LIN {X 0,Y 545.098,Z 867.396,A -85,B 0,C 180,E1 -3797.729,E2 -3797.729} C_VEL
LIN {X 0,Y 545.03,Z 867.401,A -85,B 0,C 180,E1 -3800.375,E2 -3800.375} C_VEL
LIN {X 0,Y 545.004,Z 867.406,A -85,B 0,C 180,E1 -3803.167,E2 -3803.167} C_VEL
LIN {X 0,Y 545.034,Z 867.401,A -85,B 0,C 180,E1 -3806.003,E2 -3806.003} C_VEL
LIN {X 0,Y 545.024,Z 867.401,A -85,B 0,C 180,E1 -3806.379,E2 -3806.379} C_VEL
LIN {X 0,Y 544.359,Z 867.49,A -85,B 0,C 180,E1 -3806.996,E2 -3806.996} C_VEL
LIN {X 0,Y 541.484,Z 867.844,A -85,B 0,C 180,E1 -3807.996,E2 -3807.996} C_VEL
LIN {X 0,Y 539.061,Z 868.145,A -85,B 0,C 180,E1 -3808.801,E2 -3808.801} C_VEL
LIN {X 0,Y 538.039,Z 868.281,A -85,B 0,C 180,E1 -3809.423,E2 -3809.423} C_VEL
LIN {X 0,Y 537.965,Z 868.284,A -85,B 0,C 180,E1 -3809.633,E2 -3809.633} C_VEL
LIN {X 0,Y 538.006,Z 868.275,A -85,B 0,C 180,E1 -3812.384,E2 -3812.384} C_VEL
LIN {X 0,Y 537.986,Z 868.279,A -85,B 0,C 180,E1 -3815.086,E2 -3815.086} C_VEL
LIN {X 0,Y 537.977,Z 868.281,A -85,B 0,C 180,E1 -3818.388,E2 -3818.388} C_VEL
LIN {X 0,Y 537.953,Z 868.282,A -85,B 0,C 180,E1 -3820.785,E2 -3820.785} C_VEL
LIN {X 0,Y 537.981,Z 868.284,A -85,B 0,C 180,E1 -3823.819,E2 -3823.819} C_VEL
LIN {X 0,Y 537.98,Z 868.289,A -85,B 0,C 180,E1 -3826.182,E2 -3826.182} C_VEL
LIN {X 0,Y 537.954,Z 868.281,A -85,B 0,C 180,E1 -3829.265,E2 -3829.265} C_VEL
LIN {X 0,Y 537.966,Z 868.285,A -85,B 0,C 180,E1 -3832.12,E2 -3832.12} C_VEL
LIN {X 0,Y 537.997,Z 868.277,A -85,B 0,C 180,E1 -3835.386,E2 -3835.386} C_VEL
LIN {X 0,Y 537.997,Z 868.278,A -85,B 0,C 180,E1 -3838.116,E2 -3838.116} C_VEL
LIN {X 0,Y 537.988,Z 868.284,A -85,B 0,C 180,E1 -3841.096,E2 -3841.096} C_VEL
LIN {X 0,Y 537.973,Z 868.28,A -85,B 0,C 180,E1 -3843.63,E2 -3843.63} C_VEL
LIN {X 0,Y 538.01,Z 868.274,A -85,B 0,C 180,E1 -3846.123,E2 -3846.123} C_VEL
LIN {X 0,Y 538.002,Z 868.277,A -85,B 0,C 180,E1 -3848.545,E2 -3848.545} C_VEL
LIN {X 0,Y 537.989,Z 868.281,A -85,B 0,C 180,E1 -3850.938,E2 -3850.938} C_VEL
LIN {X 0,Y 537.988,Z 868.286,A -85,B 0,C 180,E1 -3853.298,E2 -3853.298} C_VEL
LIN {X 0,Y 538.043,Z 868.278,A -85,B 0,C 180,E1 -3855.63,E2 -3855.63} C_VEL
LIN {X 0,Y 538.024,Z 868.273,A -85,B 0,C 180,E1 -3858.701,E2 -3858.701} C_VEL
LIN {X 0,Y 538.035,Z 868.281,A -85,B 0,C 180,E1 -3861.739,E2 -3861.739} C_VEL
LIN {X 0,Y 538.119,Z 868.261,A -85,B 0,C 180,E1 -3864.755,E2 -3864.755} C_VEL
LIN {X 0,Y 538.163,Z 868.261,A -85,B 0,C 180,E1 -3867.755,E2 -3867.755} C_VEL
LIN {X 0,Y 538.162,Z 868.264,A -85,B 0,C 180,E1 -3870,E2 -3870} C_VEL
LIN {X 0,Y 538.082,Z 868.266,A -85,B 0,C 180,E1 -3872.995,E2 -3872.995} C_VEL
LIN {X 0,Y 538.078,Z 868.27,A -85,B 0,C 180,E1 -3875.998,E2 -3875.998} C_VEL
LIN {X 0,Y 538.025,Z 868.276,A -85,B 0,C 180,E1 -3879.019,E2 -3879.019} C_VEL
LIN {X 0,Y 538.012,Z 868.276,A -85,B 0,C 180,E1 -3882.064,E2 -3882.064} C_VEL
LIN {X 0,Y 537.99,Z 868.282,A -85,B 0,C 180,E1 -3885.146,E2 -3885.146} C_VEL
LIN {X 0,Y 538.001,Z 868.277,A -85,B 0,C 180,E1 -3888.271,E2 -3888.271} C_VEL
LIN {X 0,Y 537.992,Z 868.281,A -85,B 0,C 180,E1 -3890.653,E2 -3890.653} C_VEL
LIN {X 0,Y 537.977,Z 868.288,A -85,B 0,C 180,E1 -3893.074,E2 -3893.074} C_VEL
LIN {X 0,Y 537.975,Z 868.283,A -85,B 0,C 180,E1 -3895.656,E2 -3895.656} C_VEL
LIN {X 0,Y 537.975,Z 868.28,A -85,B 0,C 180,E1 -3898.054,E2 -3898.054} C_VEL
LIN {X 0,Y 537.992,Z 868.277,A -85,B 0,C 180,E1 -3900.629,E2 -3900.629} C_VEL
LIN {X 0,Y 538.003,Z 868.28,A -85,B 0,C 180,E1 -3903.275,E2 -3903.275} C_VEL
LIN {X 0,Y 537.956,Z 868.287,A -85,B 0,C 180,E1 -3906.008,E2 -3906.008} C_VEL
LIN {X 0,Y 537.976,Z 868.279,A -85,B 0,C 180,E1 -3908.834,E2 -3908.834} C_VEL
LIN {X 0,Y 537.978,Z 868.287,A -85,B 0,C 180,E1 -3911.872,E2 -3911.872} C_VEL
LIN {X 0,Y 537.989,Z 868.278,A -85,B 0,C 180,E1 -3914.864,E2 -3914.864} C_VEL
LIN {X 0,Y 537.962,Z 868.28,A -85,B 0,C 180,E1 -3917.208,E2 -3917.208} C_VEL
LIN {X 0,Y 537.973,Z 868.288,A -85,B 0,C 180,E1 -3920.423,E2 -3920.423} C_VEL
LIN {X 0,Y 537.947,Z 868.284,A -85,B 0,C 180,E1 -3923.06,E2 -3923.06} C_VEL
LIN {X 0,Y 537.998,Z 868.276,A -85,B 0,C 180,E1 -3925.825,E2 -3925.825} C_VEL
LIN {X 0,Y 537.992,Z 868.283,A -85,B 0,C 180,E1 -3928.497,E2 -3928.497} C_VEL
LIN {X 0,Y 537.988,Z 868.283,A -85,B 0,C 180,E1 -3931.095,E2 -3931.095} C_VEL
LIN {X 0,Y 537.973,Z 868.28,A -85,B 0,C 180,E1 -3933.629,E2 -3933.629} C_VEL
LIN {X 0,Y 538.01,Z 868.274,A -85,B 0,C 180,E1 -3936.122,E2 -3936.122} C_VEL
LIN {X 0,Y 538.002,Z 868.277,A -85,B 0,C 180,E1 -3938.545,E2 -3938.545} C_VEL
LIN {X 0,Y 537.989,Z 868.282,A -85,B 0,C 180,E1 -3940.938,E2 -3940.938} C_VEL
LIN {X 0,Y 537.987,Z 868.286,A -85,B 0,C 180,E1 -3943.297,E2 -3943.297} C_VEL
LIN {X 0,Y 538.039,Z 868.279,A -85,B 0,C 180,E1 -3945.63,E2 -3945.63} C_VEL
LIN {X 0,Y 538.022,Z 868.273,A -85,B 0,C 180,E1 -3948.7,E2 -3948.7} C_VEL
LIN {X 0,Y 538.034,Z 868.282,A -85,B 0,C 180,E1 -3951.738,E2 -3951.738} C_VEL
LIN {X 0,Y 538.117,Z 868.261,A -85,B 0,C 180,E1 -3954.754,E2 -3954.754} C_VEL
LIN {X 0,Y 538.161,Z 868.261,A -85,B 0,C 180,E1 -3957.754,E2 -3957.754} C_VEL
LIN {X 0,Y 538.16,Z 868.264,A -85,B 0,C 180,E1 -3960,E2 -3960} C_VEL
LIN {X 0,Y 538.08,Z 868.266,A -85,B 0,C 180,E1 -3962.994,E2 -3962.994} C_VEL
LIN {X 0,Y 538.076,Z 868.27,A -85,B 0,C 180,E1 -3965.998,E2 -3965.998} C_VEL
LIN {X 0,Y 538.023,Z 868.276,A -85,B 0,C 180,E1 -3969.018,E2 -3969.018} C_VEL
LIN {X 0,Y 538.009,Z 868.276,A -85,B 0,C 180,E1 -3972.064,E2 -3972.064} C_VEL
LIN {X 0,Y 537.997,Z 868.281,A -85,B 0,C 180,E1 -3975.145,E2 -3975.145} C_VEL
LIN {X 0,Y 537.998,Z 868.277,A -85,B 0,C 180,E1 -3978.271,E2 -3978.271} C_VEL
LIN {X 0,Y 537.988,Z 868.281,A -85,B 0,C 180,E1 -3980.653,E2 -3980.653} C_VEL
LIN {X 0,Y 537.973,Z 868.288,A -85,B 0,C 180,E1 -3983.073,E2 -3983.073} C_VEL
LIN {X 0,Y 537.971,Z 868.283,A -85,B 0,C 180,E1 -3985.655,E2 -3985.655} C_VEL
LIN {X 0,Y 537.971,Z 868.28,A -85,B 0,C 180,E1 -3988.054,E2 -3988.054} C_VEL
LIN {X 0,Y 537.988,Z 868.277,A -85,B 0,C 180,E1 -3990.629,E2 -3990.629} C_VEL
LIN {X 0,Y 537.999,Z 868.281,A -85,B 0,C 180,E1 -3993.275,E2 -3993.275} C_VEL
LIN {X 0,Y 537.952,Z 868.287,A -85,B 0,C 180,E1 -3996.008,E2 -3996.008} C_VEL
LIN {X 0,Y 537.973,Z 868.279,A -85,B 0,C 180,E1 -3998.834,E2 -3998.834} C_VEL
LIN {X 0,Y 537.974,Z 868.288,A -85,B 0,C 180,E1 -4001.872,E2 -4001.872} C_VEL
LIN {X 0,Y 537.989,Z 868.278,A -85,B 0,C 180,E1 -4004.864,E2 -4004.864} C_VEL
LIN {X 0,Y 537.958,Z 868.281,A -85,B 0,C 180,E1 -4007.208,E2 -4007.208} C_VEL
LIN {X 0,Y 537.969,Z 868.289,A -85,B 0,C 180,E1 -4010.423,E2 -4010.423} C_VEL
LIN {X 0,Y 537.943,Z 868.285,A -85,B 0,C 180,E1 -4013.06,E2 -4013.06} C_VEL
LIN {X 0,Y 537.994,Z 868.277,A -85,B 0,C 180,E1 -4015.825,E2 -4015.825} C_VEL
LIN {X 0,Y 537.988,Z 868.284,A -85,B 0,C 180,E1 -4018.497,E2 -4018.497} C_VEL
LIN {X 0,Y 537.983,Z 868.284,A -85,B 0,C 180,E1 -4021.095,E2 -4021.095} C_VEL
LIN {X 0,Y 537.968,Z 868.284,A -85,B 0,C 180,E1 -4023.629,E2 -4023.629} C_VEL
LIN {X 0,Y 538.017,Z 868.284,A -85,B 0,C 180,E1 -4026.928,E2 -4026.928} C_VEL
LIN {X 0,Y 537.995,Z 868.299,A -85,B 0,C 180,E1 -4027.079,E2 -4027.079} C_VEL
LIN {X 0,Y 538.993,Z 874.286,A -85,B 0,C 180,E1 -4028.199,E2 -4028.199} C_VEL
LIN {X 0,Y 538.682,Z 889.835,A -85,B 0,C 180,E1 -4030.964,E2 -4030.964} C_VEL
LIN {X 0,Y 538.34,Z 907.701,A -85,B 0,C 180,E1 -4034.088,E2 -4034.088} C_VEL
LIN {X 0,Y 538.045,Z 925.566,A -85,B 0,C 180,E1 -4037.17,E2 -4037.17} C_VEL
LIN {X 0,Y 537.998,Z 932.73,A -85,B 0,C 180,E1 -4038.397,E2 -4038.397} C_VEL
LIN {X 0,Y 538.862,Z 941.214,A -85,B 0,C 180,E1 -4038.535,E2 -4038.535} C_VEL
LIN {X 0,Y 538.7,Z 1009.129,A -85,B 0,C 180,E1 -4039.452,E2 -4039.452} C_VEL
LIN {X 0,Y 538.545,Z 1018.405,A -85,B 0,C 180,E1 -4039.663,E2 -4039.663} C_VEL
LIN {X 0,Y 538.512,Z 1026.883,A -85,B 0,C 180,E1 -4039.947,E2 -4039.947} C_VEL
LIN {X 0,Y 538.398,Z 1035.391,A -85,B 0,C 180,E1 -4040.325,E2 -4040.325} C_VEL
LIN {X 0,Y 538.243,Z 1043.725,A -85,B 0,C 180,E1 -4040.796,E2 -4040.796} C_VEL
LIN {X 0,Y 538.128,Z 1051.765,A -85,B 0,C 180,E1 -4041.362,E2 -4041.362} C_VEL
LIN {X 0,Y 537.969,Z 1060.43,A -85,B 0,C 180,E1 -4042.116,E2 -4042.116} C_VEL
LIN {X 0,Y 537.821,Z 1068.936,A -85,B 0,C 180,E1 -4043.057,E2 -4043.057} C_VEL
LIN {X 0,Y 537.765,Z 1075.61,A -85,B 0,C 180,E1 -4043.999,E2 -4043.999} C_VEL
LIN {X 0,Y 537.605,Z 1079.988,A -85,B 0,C 180,E1 -4044.749,E2 -4044.749} C_VEL
LIN {X 0,Y 537.621,Z 1085.148,A -85,B 0,C 180,E1 -4045.877,E2 -4045.877} C_VEL
LIN {X 0,Y 537.563,Z 1088.935,A -85,B 0,C 180,E1 -4047.002,E2 -4047.002} C_VEL
LIN {X 0,Y 537.49,Z 1090.682,A -85,B 0,C 180,E1 -4047.752,E2 -4047.752} C_VEL
LIN {X 0,Y 537.45,Z 1091.933,A -85,B 0,C 180,E1 -4048.501,E2 -4048.501} C_VEL
LIN {X 0,Y 537.438,Z 1092.709,A -85,B 0,C 180,E1 -4049.251,E2 -4049.251} C_VEL
LIN {X 0,Y 537.439,Z 1093,A -85,B 0,C 180,E1 -4050,E2 -4050} C_VEL
LIN {X 0,Y 537.438,Z 1092.709,A -85,B 0,C 180,E1 -4050.749,E2 -4050.749} C_VEL
LIN {X 0,Y 537.45,Z 1091.933,A -85,B 0,C 180,E1 -4051.499,E2 -4051.499} C_VEL
LIN {X 0,Y 537.49,Z 1090.682,A -85,B 0,C 180,E1 -4052.248,E2 -4052.248} C_VEL
LIN {X 0,Y 537.588,Z 1087.788,A -85,B 0,C 180,E1 -4053.372,E2 -4053.372} C_VEL
LIN {X 0,Y 537.626,Z 1085.149,A -85,B 0,C 180,E1 -4054.123,E2 -4054.123} C_VEL
LIN {X 0,Y 537.604,Z 1079.986,A -85,B 0,C 180,E1 -4055.25,E2 -4055.25} C_VEL
LIN {X 0,Y 537.802,Z 1074.199,A -85,B 0,C 180,E1 -4056.226,E2 -4056.226} C_VEL
LIN {X 0,Y 537.852,Z 1067.437,A -85,B 0,C 180,E1 -4057.131,E2 -4057.131} C_VEL
LIN {X 0,Y 537.989,Z 1059.424,A -85,B 0,C 180,E1 -4057.978,E2 -4057.978} C_VEL
LIN {X 0,Y 538.137,Z 1051.772,A -85,B 0,C 180,E1 -4058.638,E2 -4058.638} C_VEL
LIN {X 0,Y 538.241,Z 1043.73,A -85,B 0,C 180,E1 -4059.204,E2 -4059.204} C_VEL
LIN {X 0,Y 538.398,Z 1035.398,A -85,B 0,C 180,E1 -4059.675,E2 -4059.675} C_VEL
LIN {X 0,Y 538.513,Z 1026.893,A -85,B 0,C 180,E1 -4060.053,E2 -4060.053} C_VEL
LIN {X 0,Y 538.573,Z 1016.755,A -85,B 0,C 180,E1 -4060.384,E2 -4060.384} C_VEL
LIN {X 0,Y 538.742,Z 1005.066,A -85,B 0,C 180,E1 -4060.618,E2 -4060.618} C_VEL
LIN {X 0,Y 538.73,Z 938.427,A -85,B 0,C 180,E1 -4061.505,E2 -4061.505} C_VEL
LIN {X 0,Y 537.951,Z 932.692,A -85,B 0,C 180,E1 -4061.61,E2 -4061.61} C_VEL
LIN {X 0,Y 538.174,Z 916.635,A -85,B 0,C 180,E1 -4064.366,E2 -4064.366} C_VEL
LIN {X 0,Y 538.479,Z 899.886,A -85,B 0,C 180,E1 -4067.273,E2 -4067.273} C_VEL
LIN {X 0,Y 538.838,Z 882.72,A -85,B 0,C 180,E1 -4070.295,E2 -4070.295} C_VEL
LIN {X 0,Y 538.871,Z 873.037,A -85,B 0,C 180,E1 -4072.031,E2 -4072.031} C_VEL
LIN {X 0,Y 537.994,Z 868.287,A -85,B 0,C 180,E1 -4072.92,E2 -4072.92} C_VEL
LIN {X 0,Y 537.968,Z 868.284,A -85,B 0,C 180,E1 -4075.656,E2 -4075.656} C_VEL
LIN {X 0,Y 537.968,Z 868.282,A -85,B 0,C 180,E1 -4078.054,E2 -4078.054} C_VEL
LIN {X 0,Y 537.985,Z 868.28,A -85,B 0,C 180,E1 -4080.629,E2 -4080.629} C_VEL
LIN {X 0,Y 538.018,Z 868.284,A -85,B 0,C 180,E1 -4083.278,E2 -4083.278} C_VEL
LIN {X 0,Y 537.95,Z 868.285,A -85,B 0,C 180,E1 -4086.008,E2 -4086.008} C_VEL
LIN {X 0,Y 537.97,Z 868.281,A -85,B 0,C 180,E1 -4088.834,E2 -4088.834} C_VEL
LIN {X 0,Y 537.971,Z 868.288,A -85,B 0,C 180,E1 -4091.872,E2 -4091.872} C_VEL
LIN {X 0,Y 537.983,Z 868.279,A -85,B 0,C 180,E1 -4094.865,E2 -4094.865} C_VEL
LIN {X 0,Y 537.956,Z 868.282,A -85,B 0,C 180,E1 -4097.208,E2 -4097.208} C_VEL
LIN {X 0,Y 537.968,Z 868.286,A -85,B 0,C 180,E1 -4100.424,E2 -4100.424} C_VEL
LIN {X 0,Y 537.942,Z 868.284,A -85,B 0,C 180,E1 -4103.061,E2 -4103.061} C_VEL
LIN {X 0,Y 537.993,Z 868.279,A -85,B 0,C 180,E1 -4105.825,E2 -4105.825} C_VEL
LIN {X 0,Y 537.987,Z 868.287,A -85,B 0,C 180,E1 -4108.497,E2 -4108.497} C_VEL
LIN {X 0,Y 537.983,Z 868.282,A -85,B 0,C 180,E1 -4111.096,E2 -4111.096} C_VEL
LIN {X 0,Y 537.967,Z 868.281,A -85,B 0,C 180,E1 -4113.63,E2 -4113.63} C_VEL
LIN {X 0,Y 537.981,Z 868.282,A -85,B 0,C 180,E1 -4116.129,E2 -4116.129} C_VEL
LIN {X 0,Y 537.989,Z 868.284,A -85,B 0,C 180,E1 -4118.545,E2 -4118.545} C_VEL
LIN {X 0,Y 537.986,Z 868.288,A -85,B 0,C 180,E1 -4120.938,E2 -4120.938} C_VEL
LIN {X 0,Y 538.061,Z 868.395,A -85,B 0,C 180,E1 -4122.39,E2 -4122.39} C_VEL
LIN {X 0,Y 537.938,Z 880.423,A -85,B 0,C 180,E1 -4125.192,E2 -4125.192} C_VEL
LIN {X 0,Y 537.81,Z 893.801,A -85,B 0,C 180,E1 -4128.269,E2 -4128.269} C_VEL
LIN {X 0,Y 537.801,Z 894.672,A -85,B 0,C 180,E1 -4128.468,E2 -4128.468} C_VEL
LIN {X 0,Y 538.867,Z 903.035,A -85,B 0,C 180,E1 -4128.604,E2 -4128.604} C_VEL
LIN {X 0,Y 538.651,Z 969.302,A -85,B 0,C 180,E1 -4129.499,E2 -4129.499} C_VEL
LIN {X 0,Y 538.583,Z 978.521,A -85,B 0,C 180,E1 -4129.712,E2 -4129.712} C_VEL
LIN {X 0,Y 538.444,Z 988.186,A -85,B 0,C 180,E1 -4130.041,E2 -4130.041} C_VEL
LIN {X 0,Y 538.35,Z 998.261,A -85,B 0,C 180,E1 -4130.514,E2 -4130.514} C_VEL
LIN {X 0,Y 538.217,Z 1008.735,A -85,B 0,C 180,E1 -4131.175,E2 -4131.175} C_VEL
LIN {X 0,Y 537.986,Z 1017.967,A -85,B 0,C 180,E1 -4131.927,E2 -4131.927} C_VEL
LIN {X 0,Y 537.892,Z 1025.398,A -85,B 0,C 180,E1 -4132.681,E2 -4132.681} C_VEL
LIN {X 0,Y 537.8,Z 1032.298,A -85,B 0,C 180,E1 -4133.546,E2 -4133.546} C_VEL
LIN {X 0,Y 537.652,Z 1038.788,A -85,B 0,C 180,E1 -4134.562,E2 -4134.562} C_VEL
LIN {X 0,Y 537.612,Z 1043.445,A -85,B 0,C 180,E1 -4135.502,E2 -4135.502} C_VEL
LIN {X 0,Y 537.589,Z 1047.688,A -85,B 0,C 180,E1 -4136.628,E2 -4136.628} C_VEL
LIN {X 0,Y 537.491,Z 1050.624,A -85,B 0,C 180,E1 -4137.752,E2 -4137.752} C_VEL
LIN {X 0,Y 537.45,Z 1051.926,A -85,B 0,C 180,E1 -4138.502,E2 -4138.502} C_VEL
LIN {X 0,Y 537.438,Z 1052.718,A -85,B 0,C 180,E1 -4139.251,E2 -4139.251} C_VEL
LIN {X 0,Y 537.44,Z 1052.996,A -85,B 0,C 180,E1 -4140,E2 -4140} C_VEL
LIN {X 0,Y 537.439,Z 1052.766,A -85,B 0,C 180,E1 -4140.75,E2 -4140.75} C_VEL
LIN {X 0,Y 537.451,Z 1052.038,A -85,B 0,C 180,E1 -4141.499,E2 -4141.499} C_VEL
LIN {X 0,Y 537.491,Z 1050.815,A -85,B 0,C 180,E1 -4142.248,E2 -4142.248} C_VEL
LIN {X 0,Y 537.587,Z 1047.961,A -85,B 0,C 180,E1 -4143.373,E2 -4143.373} C_VEL
LIN {X 0,Y 537.606,Z 1043.841,A -85,B 0,C 180,E1 -4144.499,E2 -4144.499} C_VEL
LIN {X 0,Y 537.71,Z 1038.231,A -85,B 0,C 180,E1 -4145.626,E2 -4145.626} C_VEL
LIN {X 0,Y 537.77,Z 1031.395,A -85,B 0,C 180,E1 -4146.671,E2 -4146.671} C_VEL
LIN {X 0,Y 537.869,Z 1024.495,A -85,B 0,C 180,E1 -4147.508,E2 -4147.508} C_VEL
LIN {X 0,Y 538.064,Z 1015.852,A -85,B 0,C 180,E1 -4148.356,E2 -4148.356} C_VEL
LIN {X 0,Y 538.275,Z 1005.984,A -85,B 0,C 180,E1 -4149.109,E2 -4149.109} C_VEL
LIN {X 0,Y 538.366,Z 996.294,A -85,B 0,C 180,E1 -4149.676,E2 -4149.676} C_VEL
LIN {X 0,Y 538.479,Z 986.822,A -85,B 0,C 180,E1 -4150.101,E2 -4150.101} C_VEL
LIN {X 0,Y 538.586,Z 976.647,A -85,B 0,C 180,E1 -4150.432,E2 -4150.432} C_VEL
LIN {X 0,Y 538.697,Z 964.837,A -85,B 0,C 180,E1 -4150.667,E2 -4150.667} C_VEL
LIN {X 0,Y 538.682,Z 900.84,A -85,B 0,C 180,E1 -4151.519,E2 -4151.519} C_VEL
LIN {X 0,Y 537.8,Z 894.627,A -85,B 0,C 180,E1 -4151.632,E2 -4151.632} C_VEL
LIN {X 0,Y 537.911,Z 882.69,A -85,B 0,C 180,E1 -4154.374,E2 -4154.374} C_VEL
LIN {X 0,Y 538.132,Z 870.991,A -85,B 0,C 180,E1 -4157.089,E2 -4157.089} C_VEL
LIN {X 0,Y 538.06,Z 868.273,A -85,B 0,C 180,E1 -4157.748,E2 -4157.748} C_VEL
LIN {X 0,Y 537.989,Z 868.281,A -85,B 0,C 180,E1 -4160.654,E2 -4160.654} C_VEL
LIN {X 0,Y 537.974,Z 868.288,A -85,B 0,C 180,E1 -4163.074,E2 -4163.074} C_VEL
LIN {X 0,Y 537.985,Z 868.282,A -85,B 0,C 180,E1 -4165.659,E2 -4165.659} C_VEL
LIN {X 0,Y 537.972,Z 868.281,A -85,B 0,C 180,E1 -4168.054,E2 -4168.054} C_VEL
LIN {X 0,Y 537.965,Z 868.284,A -85,B 0,C 180,E1 -4169.633,E2 -4169.633} C_VEL
LIN {X 0,Y 537.328,Z 868.367,A -85,B 0,C 180,E1 -4170.258,E2 -4170.258} C_VEL
LIN {X 0,Y 534.496,Z 868.718,A -85,B 0,C 180,E1 -4171.272,E2 -4171.272} C_VEL
LIN {X 0,Y 532.082,Z 869.016,A -85,B 0,C 180,E1 -4172.089,E2 -4172.089} C_VEL
LIN {X 0,Y 531.04,Z 869.143,A -85,B 0,C 180,E1 -4172.719,E2 -4172.719} C_VEL
LIN {X 0,Y 530.953,Z 869.155,A -85,B 0,C 180,E1 -4172.933,E2 -4172.933} C_VEL
LIN {X 0,Y 530.928,Z 869.165,A -85,B 0,C 180,E1 -4175.623,E2 -4175.623} C_VEL
LIN {X 0,Y 530.942,Z 869.156,A -85,B 0,C 180,E1 -4178.65,E2 -4178.65} C_VEL
LIN {X 0,Y 530.909,Z 869.161,A -85,B 0,C 180,E1 -4181.444,E2 -4181.444} C_VEL
LIN {X 0,Y 530.963,Z 869.156,A -85,B 0,C 180,E1 -4184.55,E2 -4184.55} C_VEL
LIN {X 0,Y 530.906,Z 869.16,A -85,B 0,C 180,E1 -4187.536,E2 -4187.536} C_VEL
LIN {X 0,Y 530.934,Z 869.163,A -85,B 0,C 180,E1 -4190.552,E2 -4190.552} C_VEL
LIN {X 0,Y 530.906,Z 869.159,A -85,B 0,C 180,E1 -4193.438,E2 -4193.438} C_VEL
LIN {X 0,Y 530.952,Z 869.157,A -85,B 0,C 180,E1 -4196.225,E2 -4196.225} C_VEL
LIN {X 0,Y 530.938,Z 869.163,A -85,B 0,C 180,E1 -4198.92,E2 -4198.92} C_VEL
LIN {X 0,Y 530.933,Z 869.157,A -85,B 0,C 180,E1 -4201.541,E2 -4201.541} C_VEL
LIN {X 0,Y 530.927,Z 869.157,A -85,B 0,C 180,E1 -4204.177,E2 -4204.177} C_VEL
LIN {X 0,Y 530.945,Z 869.157,A -85,B 0,C 180,E1 -4206.603,E2 -4206.603} C_VEL
LIN {X 0,Y 530.973,Z 869.159,A -85,B 0,C 180,E1 -4209.061,E2 -4209.061} C_VEL
LIN {X 0,Y 530.975,Z 869.151,A -85,B 0,C 180,E1 -4212.276,E2 -4212.276} C_VEL
LIN {X 0,Y 531.004,Z 869.157,A -85,B 0,C 180,E1 -4215.436,E2 -4215.436} C_VEL
LIN {X 0,Y 530.987,Z 869.149,A -85,B 0,C 180,E1 -4218.549,E2 -4218.549} C_VEL
LIN {X 0,Y 530.983,Z 869.158,A -85,B 0,C 180,E1 -4221.628,E2 -4221.628} C_VEL
LIN {X 0,Y 531.081,Z 869.138,A -85,B 0,C 180,E1 -4224.685,E2 -4224.685} C_VEL
LIN {X 0,Y 531.133,Z 869.136,A -85,B 0,C 180,E1 -4227.725,E2 -4227.725} C_VEL
LIN {X 0,Y 531.13,Z 869.139,A -85,B 0,C 180,E1 -4230,E2 -4230} C_VEL
LIN {X 0,Y 531.13,Z 869.141,A -85,B 0,C 180,E1 -4232.275,E2 -4232.275} C_VEL
LIN {X 0,Y 531.082,Z 869.138,A -85,B 0,C 180,E1 -4235.315,E2 -4235.315} C_VEL
LIN {X 0,Y 530.984,Z 869.158,A -85,B 0,C 180,E1 -4238.372,E2 -4238.372} C_VEL
LIN {X 0,Y 531.014,Z 869.146,A -85,B 0,C 180,E1 -4241.649,E2 -4241.649} C_VEL
LIN {X 0,Y 530.967,Z 869.16,A -85,B 0,C 180,E1 -4244.927,E2 -4244.927} C_VEL
LIN {X 0,Y 530.976,Z 869.151,A -85,B 0,C 180,E1 -4247.724,E2 -4247.724} C_VEL
LIN {X 0,Y 530.964,Z 869.16,A -85,B 0,C 180,E1 -4250.94,E2 -4250.94} C_VEL
LIN {X 0,Y 530.943,Z 869.155,A -85,B 0,C 180,E1 -4254.027,E2 -4254.027} C_VEL
LIN {X 0,Y 530.943,Z 869.157,A -85,B 0,C 180,E1 -4256.747,E2 -4256.747} C_VEL
LIN {X 0,Y 530.919,Z 869.166,A -85,B 0,C 180,E1 -4259.327,E2 -4259.327} C_VEL
LIN {X 0,Y 530.933,Z 869.159,A -85,B 0,C 180,E1 -4262.093,E2 -4262.093} C_VEL
LIN {X 0,Y 530.957,Z 869.153,A -85,B 0,C 180,E1 -4264.848,E2 -4264.848} C_VEL
LIN {X 0,Y 530.901,Z 869.166,A -85,B 0,C 180,E1 -4267.513,E2 -4267.513} C_VEL
LIN {X 0,Y 530.909,Z 869.162,A -85,B 0,C 180,E1 -4270.44,E2 -4270.44} C_VEL
LIN {X 0,Y 530.923,Z 869.159,A -85,B 0,C 180,E1 -4273.499,E2 -4273.499} C_VEL
LIN {X 0,Y 530.964,Z 869.154,A -85,B 0,C 180,E1 -4275.624,E2 -4275.624} C_VEL
LIN {X 0,Y 530.911,Z 869.165,A -85,B 0,C 180,E1 -4278.556,E2 -4278.556} C_VEL
LIN {X 0,Y 530.92,Z 869.158,A -85,B 0,C 180,E1 -4281.526,E2 -4281.526} C_VEL
LIN {X 0,Y 530.93,Z 869.164,A -85,B 0,C 180,E1 -4284.377,E2 -4284.377} C_VEL
LIN {X 0,Y 530.957,Z 869.156,A -85,B 0,C 180,E1 -4287.132,E2 -4287.132} C_VEL
LIN {X 0,Y 530.932,Z 869.156,A -85,B 0,C 180,E1 -4289.8,E2 -4289.8} C_VEL
LIN {X 0,Y 530.957,Z 869.157,A -85,B 0,C 180,E1 -4292.48,E2 -4292.48} C_VEL
LIN {X 0,Y 530.949,Z 869.155,A -85,B 0,C 180,E1 -4295.773,E2 -4295.773} C_VEL
LIN {X 0,Y 530.956,Z 869.153,A -85,B 0,C 180,E1 -4298.246,E2 -4298.246} C_VEL
LIN {X 0,Y 530.949,Z 869.156,A -85,B 0,C 180,E1 -4300.675,E2 -4300.675} C_VEL
LIN {X 0,Y 530.955,Z 869.159,A -85,B 0,C 180,E1 -4303.07,E2 -4303.07} C_VEL
LIN {X 0,Y 531.001,Z 869.158,A -85,B 0,C 180,E1 -4305.435,E2 -4305.435} C_VEL
LIN {X 0,Y 530.986,Z 869.149,A -85,B 0,C 180,E1 -4308.548,E2 -4308.548} C_VEL
LIN {X 0,Y 530.981,Z 869.158,A -85,B 0,C 180,E1 -4311.628,E2 -4311.628} C_VEL
LIN {X 0,Y 531.079,Z 869.138,A -85,B 0,C 180,E1 -4314.684,E2 -4314.684} C_VEL
LIN {X 0,Y 531.131,Z 869.137,A -85,B 0,C 180,E1 -4317.725,E2 -4317.725} C_VEL
LIN {X 0,Y 531.129,Z 869.14,A -85,B 0,C 180,E1 -4320,E2 -4320} C_VEL
LIN {X 0,Y 531.128,Z 869.141,A -85,B 0,C 180,E1 -4322.275,E2 -4322.275} C_VEL
LIN {X 0,Y 531.079,Z 869.138,A -85,B 0,C 180,E1 -4325.315,E2 -4325.315} C_VEL
LIN {X 0,Y 530.981,Z 869.158,A -85,B 0,C 180,E1 -4328.371,E2 -4328.371} C_VEL
LIN {X 0,Y 531.011,Z 869.146,A -85,B 0,C 180,E1 -4331.648,E2 -4331.648} C_VEL
LIN {X 0,Y 530.992,Z 869.156,A -85,B 0,C 180,E1 -4334.938,E2 -4334.938} C_VEL
LIN {X 0,Y 530.973,Z 869.151,A -85,B 0,C 180,E1 -4337.724,E2 -4337.724} C_VEL
LIN {X 0,Y 530.961,Z 869.161,A -85,B 0,C 180,E1 -4340.939,E2 -4340.939} C_VEL
LIN {X 0,Y 530.939,Z 869.156,A -85,B 0,C 180,E1 -4344.027,E2 -4344.027} C_VEL
LIN {X 0,Y 530.939,Z 869.157,A -85,B 0,C 180,E1 -4346.747,E2 -4346.747} C_VEL
LIN {X 0,Y 530.915,Z 869.167,A -85,B 0,C 180,E1 -4349.326,E2 -4349.326} C_VEL
LIN {X 0,Y 530.929,Z 869.159,A -85,B 0,C 180,E1 -4352.093,E2 -4352.093} C_VEL
LIN {X 0,Y 530.953,Z 869.154,A -85,B 0,C 180,E1 -4354.848,E2 -4354.848} C_VEL
LIN {X 0,Y 530.899,Z 869.166,A -85,B 0,C 180,E1 -4357.513,E2 -4357.513} C_VEL
LIN {X 0,Y 530.905,Z 869.162,A -85,B 0,C 180,E1 -4360.44,E2 -4360.44} C_VEL
LIN {X 0,Y 530.92,Z 869.16,A -85,B 0,C 180,E1 -4363.499,E2 -4363.499} C_VEL
LIN {X 0,Y 530.961,Z 869.155,A -85,B 0,C 180,E1 -4365.624,E2 -4365.624} C_VEL
LIN {X 0,Y 530.906,Z 869.165,A -85,B 0,C 180,E1 -4368.556,E2 -4368.556} C_VEL
LIN {X 0,Y 530.916,Z 869.158,A -85,B 0,C 180,E1 -4371.525,E2 -4371.525} C_VEL
LIN {X 0,Y 530.925,Z 869.165,A -85,B 0,C 180,E1 -4374.377,E2 -4374.377} C_VEL
LIN {X 0,Y 530.952,Z 869.156,A -85,B 0,C 180,E1 -4377.132,E2 -4377.132} C_VEL
LIN {X 0,Y 530.927,Z 869.157,A -85,B 0,C 180,E1 -4379.8,E2 -4379.8} C_VEL
LIN {X 0,Y 530.953,Z 869.157,A -85,B 0,C 180,E1 -4382.48,E2 -4382.48} C_VEL
LIN {X 0,Y 530.944,Z 869.16,A -85,B 0,C 180,E1 -4385.774,E2 -4385.774} C_VEL
LIN {X 0,Y 530.984,Z 869.278,A -85,B 0,C 180,E1 -4386.965,E2 -4386.965} C_VEL
LIN {X 0,Y 532.018,Z 876.369,A -85,B 0,C 180,E1 -4388.291,E2 -4388.291} C_VEL
LIN {X 0,Y 531.7,Z 892.068,A -85,B 0,C 180,E1 -4391.104,E2 -4391.104} C_VEL
LIN {X 0,Y 531.308,Z 908.817,A -85,B 0,C 180,E1 -4394.069,E2 -4394.069} C_VEL
LIN {X 0,Y 531.014,Z 925.566,A -85,B 0,C 180,E1 -4396.997,E2 -4396.997} C_VEL
LIN {X 0,Y 530.936,Z 932.708,A -85,B 0,C 180,E1 -4398.237,E2 -4398.237} C_VEL
LIN {X 0,Y 531.889,Z 940.354,A -85,B 0,C 180,E1 -4398.371,E2 -4398.371} C_VEL
LIN {X 0,Y 531.728,Z 1009.129,A -85,B 0,C 180,E1 -4399.312,E2 -4399.312} C_VEL
LIN {X 0,Y 531.588,Z 1018.405,A -85,B 0,C 180,E1 -4399.526,E2 -4399.526} C_VEL
LIN {X 0,Y 531.508,Z 1026.882,A -85,B 0,C 180,E1 -4399.813,E2 -4399.813} C_VEL
LIN {X 0,Y 531.385,Z 1035.39,A -85,B 0,C 180,E1 -4400.196,E2 -4400.196} C_VEL
LIN {X 0,Y 531.238,Z 1043.723,A -85,B 0,C 180,E1 -4400.673,E2 -4400.673} C_VEL
LIN {X 0,Y 531.099,Z 1051.763,A -85,B 0,C 180,E1 -4401.247,E2 -4401.247} C_VEL
LIN {X 0,Y 530.937,Z 1060.43,A -85,B 0,C 180,E1 -4402.011,E2 -4402.011} C_VEL
LIN {X 0,Y 530.765,Z 1068.936,A -85,B 0,C 180,E1 -4402.964,E2 -4402.964} C_VEL
LIN {X 0,Y 530.693,Z 1075.61,A -85,B 0,C 180,E1 -4403.918,E2 -4403.918} C_VEL
LIN {X 0,Y 530.542,Z 1079.988,A -85,B 0,C 180,E1 -4404.679,E2 -4404.679} C_VEL
LIN {X 0,Y 530.545,Z 1085.148,A -85,B 0,C 180,E1 -4405.822,E2 -4405.822} C_VEL
LIN {X 0,Y 530.47,Z 1088.936,A -85,B 0,C 180,E1 -4406.962,E2 -4406.962} C_VEL
LIN {X 0,Y 530.412,Z 1090.682,A -85,B 0,C 180,E1 -4407.722,E2 -4407.722} C_VEL
LIN {X 0,Y 530.359,Z 1091.932,A -85,B 0,C 180,E1 -4408.481,E2 -4408.481} C_VEL
LIN {X 0,Y 530.34,Z 1092.708,A -85,B 0,C 180,E1 -4409.241,E2 -4409.241} C_VEL
LIN {X 0,Y 530.34,Z 1093,A -85,B 0,C 180,E1 -4410,E2 -4410} C_VEL
LIN {X 0,Y 530.34,Z 1092.708,A -85,B 0,C 180,E1 -4410.759,E2 -4410.759} C_VEL
LIN {X 0,Y 530.359,Z 1091.932,A -85,B 0,C 180,E1 -4411.519,E2 -4411.519} C_VEL
LIN {X 0,Y 530.411,Z 1090.682,A -85,B 0,C 180,E1 -4412.278,E2 -4412.278} C_VEL
LIN {X 0,Y 530.494,Z 1087.787,A -85,B 0,C 180,E1 -4413.418,E2 -4413.418} C_VEL
LIN {X 0,Y 530.549,Z 1085.149,A -85,B 0,C 180,E1 -4414.178,E2 -4414.178} C_VEL
LIN {X 0,Y 530.542,Z 1079.987,A -85,B 0,C 180,E1 -4415.32,E2 -4415.32} C_VEL
LIN {X 0,Y 530.729,Z 1074.44,A -85,B 0,C 180,E1 -4416.27,E2 -4416.27} C_VEL
LIN {X 0,Y 530.793,Z 1067.436,A -85,B 0,C 180,E1 -4417.226,E2 -4417.226} C_VEL
LIN {X 0,Y 530.929,Z 1059.424,A -85,B 0,C 180,E1 -4418.085,E2 -4418.085} C_VEL
LIN {X 0,Y 531.108,Z 1051.771,A -85,B 0,C 180,E1 -4418.753,E2 -4418.753} C_VEL
LIN {X 0,Y 531.223,Z 1043.728,A -85,B 0,C 180,E1 -4419.327,E2 -4419.327} C_VEL
LIN {X 0,Y 531.384,Z 1035.396,A -85,B 0,C 180,E1 -4419.804,E2 -4419.804} C_VEL
LIN {X 0,Y 531.509,Z 1026.892,A -85,B 0,C 180,E1 -4420.186,E2 -4420.186} C_VEL
LIN {X 0,Y 531.619,Z 1016.754,A -85,B 0,C 180,E1 -4420.521,E2 -4420.521} C_VEL
LIN {X 0,Y 531.785,Z 1005.066,A -85,B 0,C 180,E1 -4420.759,E2 -4420.759} C_VEL
LIN {X 0,Y 531.736,Z 938.666,A -85,B 0,C 180,E1 -4421.655,E2 -4421.655} C_VEL
LIN {X 0,Y 530.947,Z 932.678,A -85,B 0,C 180,E1 -4421.768,E2 -4421.768} C_VEL
LIN {X 0,Y 531.175,Z 916.635,A -85,B 0,C 180,E1 -4424.56,E2 -4424.56} C_VEL
LIN {X 0,Y 531.555,Z 898.043,A -85,B 0,C 180,E1 -4427.833,E2 -4427.833} C_VEL
LIN {X 0,Y 531.846,Z 881.974,A -85,B 0,C 180,E1 -4430.708,E2 -4430.708} C_VEL
LIN {X 0,Y 531.922,Z 874.7,A -85,B 0,C 180,E1 -4431.998,E2 -4431.998} C_VEL
LIN {X 0,Y 530.983,Z 869.16,A -85,B 0,C 180,E1 -4433.034,E2 -4433.034} C_VEL
LIN {X 0,Y 530.919,Z 869.162,A -85,B 0,C 180,E1 -4435.902,E2 -4435.902} C_VEL
LIN {X 0,Y 530.927,Z 869.16,A -85,B 0,C 180,E1 -4438.46,E2 -4438.46} C_VEL
LIN {X 0,Y 530.933,Z 869.165,A -85,B 0,C 180,E1 -4441.081,E2 -4441.081} C_VEL
LIN {X 0,Y 530.947,Z 869.16,A -85,B 0,C 180,E1 -4443.776,E2 -4443.776} C_VEL
LIN {X 0,Y 530.896,Z 869.161,A -85,B 0,C 180,E1 -4446.563,E2 -4446.563} C_VEL
LIN {X 0,Y 530.928,Z 869.165,A -85,B 0,C 180,E1 -4449.449,E2 -4449.449} C_VEL
LIN {X 0,Y 530.901,Z 869.162,A -85,B 0,C 180,E1 -4452.464,E2 -4452.464} C_VEL
LIN {X 0,Y 530.956,Z 869.157,A -85,B 0,C 180,E1 -4455.45,E2 -4455.45} C_VEL
LIN {X 0,Y 530.905,Z 869.163,A -85,B 0,C 180,E1 -4458.556,E2 -4458.556} C_VEL
LIN {X 0,Y 530.916,Z 869.16,A -85,B 0,C 180,E1 -4461.526,E2 -4461.526} C_VEL
LIN {X 0,Y 530.924,Z 869.167,A -85,B 0,C 180,E1 -4464.378,E2 -4464.378} C_VEL
LIN {X 0,Y 530.951,Z 869.156,A -85,B 0,C 180,E1 -4467.133,E2 -4467.133} C_VEL
LIN {X 0,Y 530.927,Z 869.158,A -85,B 0,C 180,E1 -4469.801,E2 -4469.801} C_VEL
LIN {X 0,Y 530.952,Z 869.162,A -85,B 0,C 180,E1 -4472.48,E2 -4472.48} C_VEL
LIN {X 0,Y 530.934,Z 869.159,A -85,B 0,C 180,E1 -4475.774,E2 -4475.774} C_VEL
LIN {X 0,Y 530.946,Z 869.159,A -85,B 0,C 180,E1 -4478.246,E2 -4478.246} C_VEL
LIN {X 0,Y 530.94,Z 869.162,A -85,B 0,C 180,E1 -4480.676,E2 -4480.676} C_VEL
LIN {X 0,Y 530.995,Z 869.273,A -85,B 0,C 180,E1 -4482.356,E2 -4482.356} C_VEL
LIN {X 0,Y 530.907,Z 880.867,A -85,B 0,C 180,E1 -4485.095,E2 -4485.095} C_VEL
LIN {X 0,Y 530.737,Z 894.708,A -85,B 0,C 180,E1 -4488.314,E2 -4488.314} C_VEL
LIN {X 0,Y 531.904,Z 902.44,A -85,B 0,C 180,E1 -4488.444,E2 -4488.444} C_VEL
LIN {X 0,Y 531.693,Z 969.335,A -85,B 0,C 180,E1 -4489.36,E2 -4489.36} C_VEL
LIN {X 0,Y 531.622,Z 978.541,A -85,B 0,C 180,E1 -4489.575,E2 -4489.575} C_VEL
LIN {X 0,Y 531.461,Z 988.199,A -85,B 0,C 180,E1 -4489.909,E2 -4489.909} C_VEL
LIN {X 0,Y 531.357,Z 998.276,A -85,B 0,C 180,E1 -4490.388,E2 -4490.388} C_VEL
LIN {X 0,Y 531.206,Z 1008.738,A -85,B 0,C 180,E1 -4491.057,E2 -4491.057} C_VEL
LIN {X 0,Y 530.95,Z 1017.976,A -85,B 0,C 180,E1 -4491.82,E2 -4491.82} C_VEL
LIN {X 0,Y 530.832,Z 1025.409,A -85,B 0,C 180,E1 -4492.584,E2 -4492.584} C_VEL
LIN {X 0,Y 530.714,Z 1032.835,A -85,B 0,C 180,E1 -4493.536,E2 -4493.536} C_VEL
LIN {X 0,Y 530.597,Z 1038.791,A -85,B 0,C 180,E1 -4494.49,E2 -4494.49} C_VEL
LIN {X 0,Y 530.514,Z 1043.444,A -85,B 0,C 180,E1 -4495.441,E2 -4495.441} C_VEL
LIN {X 0,Y 530.496,Z 1047.693,A -85,B 0,C 180,E1 -4496.583,E2 -4496.583} C_VEL
LIN {X 0,Y 530.412,Z 1050.629,A -85,B 0,C 180,E1 -4497.722,E2 -4497.722} C_VEL
LIN {X 0,Y 530.359,Z 1051.931,A -85,B 0,C 180,E1 -4498.482,E2 -4498.482} C_VEL
LIN {X 0,Y 530.34,Z 1052.718,A -85,B 0,C 180,E1 -4499.241,E2 -4499.241} C_VEL
LIN {X 0,Y 530.341,Z 1052.997,A -85,B 0,C 180,E1 -4500,E2 -4500} C_VEL
LIN {X 0,Y 530.341,Z 1052.769,A -85,B 0,C 180,E1 -4500.76,E2 -4500.76} C_VEL
LIN {X 0,Y 530.361,Z 1052.042,A -85,B 0,C 180,E1 -4501.519,E2 -4501.519} C_VEL
LIN {X 0,Y 530.413,Z 1050.818,A -85,B 0,C 180,E1 -4502.278,E2 -4502.278} C_VEL
LIN {X 0,Y 530.494,Z 1047.961,A -85,B 0,C 180,E1 -4503.418,E2 -4503.418} C_VEL
LIN {X 0,Y 530.507,Z 1043.836,A -85,B 0,C 180,E1 -4504.559,E2 -4504.559} C_VEL
LIN {X 0,Y 530.658,Z 1038.228,A -85,B 0,C 180,E1 -4505.701,E2 -4505.701} C_VEL
LIN {X 0,Y 530.693,Z 1032.026,A -85,B 0,C 180,E1 -4506.671,E2 -4506.671} C_VEL
LIN {X 0,Y 530.833,Z 1024.487,A -85,B 0,C 180,E1 -4507.608,E2 -4507.608} C_VEL
LIN {X 0,Y 531.028,Z 1015.844,A -85,B 0,C 180,E1 -4508.467,E2 -4508.467} C_VEL
LIN {X 0,Y 531.258,Z 1005.975,A -85,B 0,C 180,E1 -4509.231,E2 -4509.231} C_VEL
LIN {X 0,Y 531.357,Z 996.278,A -85,B 0,C 180,E1 -4509.805,E2 -4509.805} C_VEL
LIN {X 0,Y 531.479,Z 986.804,A -85,B 0,C 180,E1 -4510.236,E2 -4510.236} C_VEL
LIN {X 0,Y 531.622,Z 976.624,A -85,B 0,C 180,E1 -4510.57,E2 -4510.57} C_VEL
LIN {X 0,Y 531.737,Z 964.792,A -85,B 0,C 180,E1 -4510.808,E2 -4510.808} C_VEL
LIN {X 0,Y 531.729,Z 901.471,A -85,B 0,C 180,E1 -4511.662,E2 -4511.662} C_VEL
LIN {X 0,Y 530.725,Z 894.572,A -85,B 0,C 180,E1 -4511.802,E2 -4511.802} C_VEL
LIN {X 0,Y 530.908,Z 881.248,A -85,B 0,C 180,E1 -4514.905,E2 -4514.905} C_VEL
LIN {X 0,Y 531.065,Z 869.542,A -85,B 0,C 180,E1 -4517.668,E2 -4517.668} C_VEL
LIN {X 0,Y 531.038,Z 869.148,A -85,B 0,C 180,E1 -4517.822,E2 -4517.822} C_VEL
LIN {X 0,Y 530.961,Z 869.16,A -85,B 0,C 180,E1 -4520.94,E2 -4520.94} C_VEL
LIN {X 0,Y 530.952,Z 869.154,A -85,B 0,C 180,E1 -4524.031,E2 -4524.031} C_VEL
LIN {X 0,Y 530.945,Z 869.156,A -85,B 0,C 180,E1 -4526.747,E2 -4526.747} C_VEL
LIN {X 0,Y 530.907,Z 869.163,A -85,B 0,C 180,E1 -4529.633,E2 -4529.633} C_VEL
LIN {X 0,Y 530.953,Z 869.156,A -85,B 0,C 180,E1 -4532.098,E2 -4532.098} C_VEL
LIN {X 0,Y 530.953,Z 869.155,A -85,B 0,C 180,E1 -4532.933,E2 -4532.933} C_VEL
LIN {X 0,Y 530.274,Z 869.247,A -85,B 0,C 180,E1 -4533.566,E2 -4533.566} C_VEL
LIN {X 0,Y 527.392,Z 869.607,A -85,B 0,C 180,E1 -4534.595,E2 -4534.595} C_VEL
LIN {X 0,Y 524.967,Z 869.908,A -85,B 0,C 180,E1 -4535.423,E2 -4535.423} C_VEL
LIN {X 0,Y 523.936,Z 870.033,A -85,B 0,C 180,E1 -4536.063,E2 -4536.063} C_VEL
LIN {X 0,Y 523.856,Z 870.04,A -85,B 0,C 180,E1 -4536.279,E2 -4536.279} C_VEL
LIN {X 0,Y 523.894,Z 870.033,A -85,B 0,C 180,E1 -4539.088,E2 -4539.088} C_VEL
LIN {X 0,Y 523.875,Z 870.039,A -85,B 0,C 180,E1 -4542.452,E2 -4542.452} C_VEL
LIN {X 0,Y 523.933,Z 870.028,A -85,B 0,C 180,E1 -4545.312,E2 -4545.312} C_VEL
LIN {X 0,Y 523.878,Z 870.039,A -85,B 0,C 180,E1 -4548.7,E2 -4548.7} C_VEL
LIN {X 0,Y 523.884,Z 870.036,A -85,B 0,C 180,E1 -4551.895,E2 -4551.895} C_VEL
LIN {X 0,Y 523.916,Z 870.035,A -85,B 0,C 180,E1 -4554.914,E2 -4554.914} C_VEL
LIN {X 0,Y 523.903,Z 870.032,A -85,B 0,C 180,E1 -4557.686,E2 -4557.686} C_VEL
LIN {X 0,Y 523.868,Z 870.038,A -85,B 0,C 180,E1 -4560.239,E2 -4560.239} C_VEL
LIN {X 0,Y 523.894,Z 870.042,A -85,B 0,C 180,E1 -4562.864,E2 -4562.864} C_VEL
LIN {X 0,Y 523.914,Z 870.031,A -85,B 0,C 180,E1 -4565.81,E2 -4565.81} C_VEL
LIN {X 0,Y 523.926,Z 870.032,A -85,B 0,C 180,E1 -4568.766,E2 -4568.766} C_VEL
LIN {X 0,Y 523.919,Z 870.039,A -85,B 0,C 180,E1 -4571.22,E2 -4571.22} C_VEL
LIN {X 0,Y 523.893,Z 870.039,A -85,B 0,C 180,E1 -4573.638,E2 -4573.638} C_VEL
LIN {X 0,Y 523.916,Z 870.033,A -85,B 0,C 180,E1 -4576.027,E2 -4576.027} C_VEL
LIN {X 0,Y 523.962,Z 870.025,A -85,B 0,C 180,E1 -4578.393,E2 -4578.393} C_VEL
LIN {X 0,Y 523.947,Z 870.032,A -85,B 0,C 180,E1 -4581.515,E2 -4581.515} C_VEL
LIN {X 0,Y 524.006,Z 870.029,A -85,B 0,C 180,E1 -4583.841,E2 -4583.841} C_VEL
LIN {X 0,Y 524.102,Z 870.012,A -85,B 0,C 180,E1 -4587.695,E2 -4587.695} C_VEL
LIN {X 0,Y 524.099,Z 870.015,A -85,B 0,C 180,E1 -4590,E2 -4590} C_VEL
LIN {X 0,Y 524.1,Z 870.016,A -85,B 0,C 180,E1 -4592.306,E2 -4592.306} C_VEL
LIN {X 0,Y 524.003,Z 870.025,A -85,B 0,C 180,E1 -4596.16,E2 -4596.16} C_VEL
LIN {X 0,Y 523.943,Z 870.028,A -85,B 0,C 180,E1 -4599.263,E2 -4599.263} C_VEL
LIN {X 0,Y 523.923,Z 870.035,A -85,B 0,C 180,E1 -4602.394,E2 -4602.394} C_VEL
LIN {X 0,Y 523.889,Z 870.034,A -85,B 0,C 180,E1 -4605.563,E2 -4605.563} C_VEL
LIN {X 0,Y 523.915,Z 870.03,A -85,B 0,C 180,E1 -4607.971,E2 -4607.971} C_VEL
LIN {X 0,Y 523.926,Z 870.03,A -85,B 0,C 180,E1 -4610.412,E2 -4610.412} C_VEL
LIN {X 0,Y 523.887,Z 870.04,A -85,B 0,C 180,E1 -4612.895,E2 -4612.895} C_VEL
LIN {X 0,Y 523.875,Z 870.043,A -85,B 0,C 180,E1 -4615.423,E2 -4615.423} C_VEL
LIN {X 0,Y 523.9,Z 870.034,A -85,B 0,C 180,E1 -4618.003,E2 -4618.003} C_VEL
LIN {X 0,Y 523.899,Z 870.034,A -85,B 0,C 180,E1 -4620.845,E2 -4620.845} C_VEL
LIN {X 0,Y 523.915,Z 870.039,A -85,B 0,C 180,E1 -4623.726,E2 -4623.726} C_VEL
LIN {X 0,Y 523.858,Z 870.039,A -85,B 0,C 180,E1 -4626.394,E2 -4626.394} C_VEL
LIN {X 0,Y 523.89,Z 870.034,A -85,B 0,C 180,E1 -4629.088,E2 -4629.088} C_VEL
LIN {X 0,Y 523.89,Z 870.041,A -85,B 0,C 180,E1 -4632.125,E2 -4632.125} C_VEL
LIN {X 0,Y 523.933,Z 870.028,A -85,B 0,C 180,E1 -4635.312,E2 -4635.312} C_VEL
LIN {X 0,Y 523.879,Z 870.039,A -85,B 0,C 180,E1 -4638.7,E2 -4638.7} C_VEL
LIN {X 0,Y 523.876,Z 870.037,A -85,B 0,C 180,E1 -4641.894,E2 -4641.894} C_VEL
LIN {X 0,Y 523.917,Z 870.035,A -85,B 0,C 180,E1 -4644.913,E2 -4644.913} C_VEL
LIN {X 0,Y 523.904,Z 870.032,A -85,B 0,C 180,E1 -4647.686,E2 -4647.686} C_VEL
LIN {X 0,Y 523.869,Z 870.038,A -85,B 0,C 180,E1 -4650.239,E2 -4650.239} C_VEL
LIN {X 0,Y 523.894,Z 870.042,A -85,B 0,C 180,E1 -4652.863,E2 -4652.863} C_VEL
LIN {X 0,Y 523.914,Z 870.031,A -85,B 0,C 180,E1 -4655.809,E2 -4655.809} C_VEL
LIN {X 0,Y 523.926,Z 870.033,A -85,B 0,C 180,E1 -4658.765,E2 -4658.765} C_VEL
LIN {X 0,Y 523.919,Z 870.039,A -85,B 0,C 180,E1 -4661.219,E2 -4661.219} C_VEL
LIN {X 0,Y 523.89,Z 870.039,A -85,B 0,C 180,E1 -4663.637,E2 -4663.637} C_VEL
LIN {X 0,Y 523.911,Z 870.033,A -85,B 0,C 180,E1 -4666.027,E2 -4666.027} C_VEL
LIN {X 0,Y 523.961,Z 870.025,A -85,B 0,C 180,E1 -4668.393,E2 -4668.393} C_VEL
LIN {X 0,Y 523.945,Z 870.033,A -85,B 0,C 180,E1 -4671.515,E2 -4671.515} C_VEL
LIN {X 0,Y 524.005,Z 870.029,A -85,B 0,C 180,E1 -4673.84,E2 -4673.84} C_VEL
LIN {X 0,Y 524.1,Z 870.012,A -85,B 0,C 180,E1 -4677.694,E2 -4677.694} C_VEL
LIN {X 0,Y 524.097,Z 870.016,A -85,B 0,C 180,E1 -4680,E2 -4680} C_VEL
LIN {X 0,Y 524.098,Z 870.016,A -85,B 0,C 180,E1 -4682.305,E2 -4682.305} C_VEL
LIN {X 0,Y 524.001,Z 870.026,A -85,B 0,C 180,E1 -4686.159,E2 -4686.159} C_VEL
LIN {X 0,Y 523.94,Z 870.028,A -85,B 0,C 180,E1 -4689.263,E2 -4689.263} C_VEL
LIN {X 0,Y 523.921,Z 870.035,A -85,B 0,C 180,E1 -4692.393,E2 -4692.393} C_VEL
LIN {X 0,Y 523.943,Z 870.033,A -85,B 0,C 180,E1 -4695.03,E2 -4695.03} C_VEL
